   LIN {X -3.366, Y 22.640, Z 44.200}
   LaserEnd_Ext()
   LIN {X 4.267, Y 22.640, Z 44.200}
   LaserStart_Ext()
   LIN {X 6.316, Y 22.640, Z 44.200}
   LaserEnd_Ext()
   LIN {X 6.105, Y 23.640, Z 44.200}
   LaserStart_Ext()
   LIN {X 4.185, Y 23.640, Z 44.200}
   LaserEnd_Ext()
   LIN {X -3.448, Y 23.640, Z 44.200}
   LaserStart_Ext()
   LIN {X -5.428, Y 23.640, Z 44.200}
   LaserEnd_Ext()
   LIN {X -5.387, Y 24.640, Z 44.200}
   LaserStart_Ext()
   LIN {X -3.576, Y 24.640, Z 44.200}
   LaserEnd_Ext()
   LIN {X 4.102, Y 24.640, Z 44.200}
   LaserStart_Ext()
   LIN {X 5.868, Y 24.640, Z 44.200}
   LaserEnd_Ext()
   LIN {X 5.630, Y 25.640, Z 44.200}
   LaserStart_Ext()
   LIN {X 4.020, Y 25.640, Z 44.200}
   LaserEnd_Ext()
   LIN {X -3.712, Y 25.640, Z 44.200}
   LaserStart_Ext()
   LIN {X -5.345, Y 25.640, Z 44.200}
   LaserEnd_Ext()
   LIN {X -5.304, Y 26.640, Z 44.200}
   LaserStart_Ext()
   LIN {X -3.861, Y 26.640, Z 44.200}
   LaserEnd_Ext()
   LIN {X 3.938, Y 26.640, Z 44.200}
   LaserStart_Ext()
   LIN {X 5.393, Y 26.640, Z 44.200}
   LaserEnd_Ext()
   LIN {X 5.155, Y 27.640, Z 44.200}
   LaserStart_Ext()
   LIN {X 3.855, Y 27.640, Z 44.200}
   LaserEnd_Ext()
   LIN {X -4.010, Y 27.640, Z 44.200}
   LaserStart_Ext()
   LIN {X -5.263, Y 27.640, Z 44.200}
   LaserEnd_Ext()
   LIN {X -5.222, Y 28.640, Z 44.200}
   LaserStart_Ext()
   LIN {X -4.204, Y 28.640, Z 44.200}
   LaserEnd_Ext()
   LIN {X 3.773, Y 28.640, Z 44.200}
   LaserStart_Ext()
   LIN {X 4.911, Y 28.640, Z 44.200}
   LaserEnd_Ext()
   LIN {X 4.626, Y 29.640, Z 44.200}
   LaserStart_Ext()
   LIN {X 3.690, Y 29.640, Z 44.200}
   LaserEnd_Ext()
   LIN {X -4.407, Y 29.640, Z 44.200}
   LaserStart_Ext()
   LIN {X -5.180, Y 29.640, Z 44.200}
   LaserEnd_Ext()
   LIN {X -5.139, Y 30.640, Z 44.200}
   LaserStart_Ext()
   LIN {X -4.596, Y 30.640, Z 44.200}
   LaserEnd_Ext()
   LIN {X 3.608, Y 30.640, Z 44.200}
   LaserStart_Ext()
   LIN {X 4.336, Y 30.640, Z 44.200}
   LaserEnd_Ext()
   LIN {X 4.045, Y 31.640, Z 44.200}
   LaserStart_Ext()
   LIN {X 3.526, Y 31.640, Z 44.200}
   LaserEnd_Ext()
   LIN {X -4.818, Y 31.640, Z 44.200}
   LaserStart_Ext()
   LIN {X -5.098, Y 31.640, Z 44.200}
   LaserEnd_Ext()
   LIN {X 3.443, Y 32.640, Z 44.200}
   LaserStart_Ext()
   LIN {X 3.755, Y 32.640, Z 44.200}
   LaserEnd_Ext()
   LIN {X 3.446, Y 33.640, Z 44.200}
   LaserStart_Ext()
   LIN {X 3.361, Y 33.640, Z 44.200}
   LaserEnd_Ext()
   LIN {X -4.883, Y 40.640, Z 44.200}
   LaserStart_Ext()
   LIN {X -4.510, Y 40.640, Z 44.200}
   LaserEnd_Ext()
   LIN {X -1.332, Y 41.640, Z 44.200}
   LaserStart_Ext()
   LIN {X -4.514, Y 41.640, Z 44.200}
   LaserEnd_Ext()
   LIN {X -3.132, Y 42.640, Z 44.200}
   LaserStart_Ext()
   LIN {X -0.665, Y 42.640, Z 44.200}
   LaserEnd_Ext()
   LIN {X -6.671, Y -21.178, Z 45.050}
   LaserStart_Ext()
   LIN {X -6.610, Y -21.017, Z 45.050} C_DIS
   LIN {X -5.679, Y -18.475, Z 45.050} C_DIS
   LIN {X -4.713, Y -17.579, Z 45.050} C_DIS
   LIN {X -4.214, Y -17.153, Z 45.050} C_DIS
   LIN {X -3.553, Y -16.965, Z 45.050} C_DIS
   LIN {X -1.903, Y -16.452, Z 45.050} C_DIS
   LIN {X 0.145, Y -16.770, Z 45.050} C_DIS
   LIN {X 0.270, Y -16.853, Z 45.050} C_DIS
   LIN {X 1.918, Y -17.941, Z 45.050} C_DIS
   LIN {X 3.157, Y -20.130, Z 45.050} C_DIS
   LIN {X 3.247, Y -22.329, Z 45.050} C_DIS
   LIN {X 2.840, Y -23.310, Z 45.050} C_DIS
   LIN {X 2.329, Y -24.417, Z 45.050} C_DIS
   LIN {X 1.031, Y -25.558, Z 45.050} C_DIS
   LIN {X 0.668, Y -25.856, Z 45.050} C_DIS
   LIN {X -0.475, Y -26.166, Z 45.050} C_DIS
   LIN {X -1.451, Y -26.443, Z 45.050} C_DIS
   LIN {X -1.877, Y -26.384, Z 45.050} C_DIS
   LIN {X -3.505, Y -26.122, Z 45.050} C_DIS
   LIN {X -5.111, Y -25.071, Z 45.050} C_DIS
   LIN {X -5.233, Y -24.991, Z 45.050} C_DIS
   LIN {X -5.333, Y -24.835, Z 45.050} C_DIS
   LIN {X -6.364, Y -23.242, Z 45.050} C_DIS
   LIN {X -6.654, Y -21.290, Z 45.050} C_DIS
   LIN {X -6.671, Y -21.178, Z 45.050}
   LaserEnd_Ext()
   LIN {X 2.040, Y 40.494, Z 45.050}
   LaserStart_Ext()
   LIN {X 1.604, Y 41.595, Z 45.050} C_DIS
   LIN {X 0.827, Y 42.817, Z 45.050} C_DIS
   LIN {X -0.621, Y 43.824, Z 45.050} C_DIS
   LIN {X -1.693, Y 44.003, Z 45.050} C_DIS
   LIN {X -2.344, Y 44.109, Z 45.050} C_DIS
   LIN {X -4.381, Y 43.298, Z 45.050} C_DIS
   LIN {X -4.665, Y 43.190, Z 45.050} C_DIS
   LIN {X -5.200, Y 42.535, Z 45.050} C_DIS
   LIN {X -5.616, Y 42.020, Z 45.050} C_DIS
   LIN {X -5.782, Y 41.406, Z 45.050} C_DIS
   LIN {X -6.083, Y 40.281, Z 45.050} C_DIS
   LIN {X -6.024, Y 39.918, Z 45.050} C_DIS
   LIN {X -5.867, Y 38.846, Z 45.050} C_DIS
   LIN {X -5.515, Y 37.770, Z 45.050} C_DIS
   LIN {X -5.478, Y 37.657, Z 45.050} C_DIS
   LIN {X -5.400, Y 37.403, Z 45.050} C_DIS
   LIN {X -5.004, Y 36.129, Z 45.050} C_DIS
   LIN {X -4.447, Y 34.142, Z 45.050} C_DIS
   LIN {X -4.364, Y 33.846, Z 45.050} C_DIS
   LIN {X -4.275, Y 33.476, Z 45.050} C_DIS
   LIN {X -3.760, Y 31.370, Z 45.050} C_DIS
   LIN {X -3.599, Y 30.520, Z 45.050} C_DIS
   LIN {X -3.113, Y 28.175, Z 45.050} C_DIS
   LIN {X -2.524, Y 24.212, Z 45.050} C_DIS
   LIN {X -2.413, Y 23.341, Z 45.050} C_DIS
   LIN {X -2.410, Y 22.832, Z 45.050} C_DIS
   LIN {X -1.992, Y 12.633, Z 45.050} C_DIS
   LIN {X -2.507, Y 7.770, Z 45.050} C_DIS
   LIN {X -2.774, Y 4.413, Z 45.050} C_DIS
   LIN {X -2.802, Y 4.238, Z 45.050} C_DIS
   LIN {X -3.922, Y -1.528, Z 45.050} C_DIS
   LIN {X -4.521, Y -3.749, Z 45.050} C_DIS
   LIN {X -5.169, Y -6.114, Z 45.050} C_DIS
   LIN {X -5.915, Y -8.275, Z 45.050} C_DIS
   LIN {X -6.675, Y -10.509, Z 45.050} C_DIS
   LIN {X -7.437, Y -12.386, Z 45.050} C_DIS
   LIN {X -8.086, Y -13.961, Z 45.050} C_DIS
   LIN {X -9.001, Y -15.896, Z 45.050} C_DIS
   LIN {X -9.722, Y -17.441, Z 45.050} C_DIS
   LIN {X -10.005, Y -18.403, Z 45.050} C_DIS
   LIN {X -10.631, Y -20.479, Z 45.050} C_DIS
   LIN {X -10.320, Y -23.787, Z 45.050} C_DIS
   LIN {X -10.287, Y -24.174, Z 45.050} C_DIS
   LIN {X -10.044, Y -24.611, Z 45.050} C_DIS
   LIN {X -8.449, Y -27.442, Z 45.050} C_DIS
   LIN {X -7.017, Y -28.613, Z 45.050} C_DIS
   LIN {X -6.195, Y -29.276, Z 45.050} C_DIS
   LIN {X -5.563, Y -29.496, Z 45.050} C_DIS
   LIN {X -2.915, Y -30.379, Z 45.050} C_DIS
   LIN {X -0.191, Y -30.129, Z 45.050} C_DIS
   LIN {X 1.018, Y -30.030, Z 45.050} C_DIS
   LIN {X 3.540, Y -28.664, Z 45.050} C_DIS
   LIN {X 3.985, Y -28.426, Z 45.050} C_DIS
   LIN {X 4.171, Y -28.214, Z 45.050} C_DIS
   LIN {X 5.934, Y -26.228, Z 45.050} C_DIS
   LIN {X 6.828, Y -24.050, Z 45.050} C_DIS
   LIN {X 7.136, Y -23.314, Z 45.050} C_DIS
   LIN {X 7.378, Y -22.094, Z 45.050} C_DIS
   LIN {X 7.781, Y -20.115, Z 45.050} C_DIS
   LIN {X 8.099, Y -18.306, Z 45.050} C_DIS
   LIN {X 8.287, Y -17.198, Z 45.050} C_DIS
   LIN {X 8.496, Y -15.692, Z 45.050} C_DIS
   LIN {X 8.821, Y -13.430, Z 45.050} C_DIS
   LIN {X 9.039, Y -11.387, Z 45.050} C_DIS
   LIN {X 9.307, Y -8.680, Z 45.050} C_DIS
   LIN {X 9.533, Y -4.472, Z 45.050} C_DIS
   LIN {X 9.615, Y -3.097, Z 45.050} C_DIS
   LIN {X 9.614, Y -1.693, Z 45.050} C_DIS
   LIN {X 9.577, Y 4.772, Z 45.050} C_DIS
   LIN {X 9.079, Y 9.376, Z 45.050} C_DIS
   LIN {X 8.618, Y 14.785, Z 45.050} C_DIS
   LIN {X 7.738, Y 20.619, Z 45.050} C_DIS
   LIN {X 6.990, Y 24.194, Z 45.050} C_DIS
   LIN {X 6.003, Y 28.349, Z 45.050} C_DIS
   LIN {X 5.310, Y 30.781, Z 45.050} C_DIS
   LIN {X 4.593, Y 33.246, Z 45.050} C_DIS
   LIN {X 4.021, Y 34.987, Z 45.050} C_DIS
   LIN {X 3.789, Y 35.696, Z 45.050} C_DIS
   LIN {X 3.724, Y 35.896, Z 45.050} C_DIS
   LIN {X 3.403, Y 36.808, Z 45.050} C_DIS
   LIN {X 2.943, Y 38.106, Z 45.050} C_DIS
   LIN {X 2.431, Y 39.464, Z 45.050} C_DIS
   LIN {X 2.153, Y 40.206, Z 45.050} C_DIS
   LIN {X 2.040, Y 40.494, Z 45.050}
   LaserEnd_Ext()
   LIN {X 8.602, Y 0.379, Z 45.050}
   LaserStart_Ext()
   LIN {X 8.602, Y -3.288, Z 45.050}
   LaserEnd_Ext()
   LIN {X 7.602, Y -14.881, Z 45.050}
   LaserStart_Ext()
   LIN {X 7.602, Y 14.818, Z 45.050}
   LaserEnd_Ext()
   LIN {X 6.602, Y 21.165, Z 45.050}
   LaserStart_Ext()
   LIN {X 6.602, Y -20.894, Z 45.050}
   LaserEnd_Ext()
   LIN {X 5.602, Y -24.403, Z 45.050}
   LaserStart_Ext()
   LIN {X 5.602, Y 25.712, Z 45.050}
   LaserEnd_Ext()
   LIN {X 4.602, Y 29.617, Z 45.050}
   LaserStart_Ext()
   LIN {X 4.602, Y -26.222, Z 45.050}
   LaserEnd_Ext()
   LIN {X 3.602, Y -27.349, Z 45.050}
   LaserStart_Ext()
   LIN {X 3.602, Y -24.045, Z 45.050}
   LaserEnd_Ext()
   LIN {X 3.602, Y -18.886, Z 45.050}
   LaserStart_Ext()
   LIN {X 3.602, Y 33.060, Z 45.050}
   LaserEnd_Ext()
   LIN {X 2.602, Y 36.071, Z 45.050}
   LaserStart_Ext()
   LIN {X 2.602, Y -17.212, Z 45.050}
   LaserEnd_Ext()
   LIN {X 2.602, Y -25.509, Z 45.050}
   LaserStart_Ext()
   LIN {X 2.602, Y -28.034, Z 45.050}
   LaserEnd_Ext()
   LIN {X 1.602, Y -28.576, Z 45.050}
   LaserStart_Ext()
   LIN {X 1.602, Y -26.383, Z 45.050}
   LaserEnd_Ext()
   LIN {X 1.602, Y -16.534, Z 45.050}
   LaserStart_Ext()
   LIN {X 1.602, Y 38.829, Z 45.050}
   LaserEnd_Ext()
   LIN {X 0.602, Y 41.307, Z 45.050}
   LaserStart_Ext()
   LIN {X 0.602, Y -15.881, Z 45.050}
   LaserEnd_Ext()
   LIN {X 0.602, Y -26.910, Z 45.050}
   LaserStart_Ext()
   LIN {X 0.602, Y -29.061, Z 45.050}
   LaserEnd_Ext()
   LIN {X -0.398, Y -29.144, Z 45.050}
   LaserStart_Ext()
   LIN {X -0.398, Y -27.184, Z 45.050}
   LaserEnd_Ext()
   LIN {X -0.398, Y -15.673, Z 45.050}
   LaserStart_Ext()
   LIN {X -0.398, Y 42.457, Z 45.050}
   LaserEnd_Ext()
   LIN {X -1.398, Y 42.940, Z 45.050}
   LaserStart_Ext()
   LIN {X -1.398, Y 22.553, Z 45.050}
   LaserEnd_Ext()
   LIN {X -1.398, Y 8.750, Z 45.050}
   LaserStart_Ext()
   LIN {X -1.398, Y -15.518, Z 45.050}
   LaserEnd_Ext()
   LIN {X -1.398, Y -27.441, Z 45.050}
   LaserStart_Ext()
   LIN {X -1.398, Y -29.235, Z 45.050}
   LaserEnd_Ext()
   LIN {X -2.398, Y -29.327, Z 45.050}
   LaserStart_Ext()
   LIN {X -2.398, Y -27.313, Z 45.050}
   LaserEnd_Ext()
   LIN {X -2.398, Y -15.558, Z 45.050}
   LaserStart_Ext()
   LIN {X -2.398, Y 1.074, Z 45.050}
   LaserEnd_Ext()
   LIN {X -2.398, Y 29.651, Z 45.050}
   LaserStart_Ext()
   LIN {X -2.398, Y 43.011, Z 45.050}
   LaserEnd_Ext()
   LIN {X -3.398, Y 42.613, Z 45.050}
   LaserStart_Ext()
   LIN {X -3.398, Y 34.104, Z 45.050}
   LaserEnd_Ext()
   LIN {X -3.398, Y -3.425, Z 45.050}
   LaserStart_Ext()
   LIN {X -3.398, Y -15.869, Z 45.050}
   LaserEnd_Ext()
   LIN {X -3.398, Y -27.152, Z 45.050}
   LaserStart_Ext()
   LIN {X -3.398, Y -29.164, Z 45.050}
   LaserEnd_Ext()
   LIN {X -4.398, Y -28.831, Z 45.050}
   LaserStart_Ext()
   LIN {X -4.398, Y -26.732, Z 45.050}
   LaserEnd_Ext()
   LIN {X -4.398, Y -16.166, Z 45.050}
   LaserStart_Ext()
   LIN {X -4.398, Y -6.945, Z 45.050}
   LaserEnd_Ext()
   LIN {X -4.398, Y 37.549, Z 45.050}
   LaserStart_Ext()
   LIN {X -4.398, Y 41.937, Z 45.050}
   LaserEnd_Ext()
   LIN {X -5.398, Y -9.861, Z 45.050}
   LaserStart_Ext()
   LIN {X -5.398, Y -16.851, Z 45.050}
   LaserEnd_Ext()
   LIN {X -5.398, Y -26.078, Z 45.050}
   LaserStart_Ext()
   LIN {X -5.398, Y -28.495, Z 45.050}
   LaserEnd_Ext()
   LIN {X -6.398, Y -27.827, Z 45.050}
   LaserStart_Ext()
   LIN {X -6.398, Y -25.029, Z 45.050}
   LaserEnd_Ext()
   LIN {X -6.398, Y -17.782, Z 45.050}
   LaserStart_Ext()
   LIN {X -6.398, Y -12.485, Z 45.050}
   LaserEnd_Ext()
   LIN {X -7.398, Y -14.846, Z 45.050}
   LaserStart_Ext()
   LIN {X -7.398, Y -20.261, Z 45.050}
   LaserEnd_Ext()
   LIN {X -7.398, Y -23.085, Z 45.050}
   LaserStart_Ext()
   LIN {X -7.398, Y -27.010, Z 45.050}
   LaserEnd_Ext()
   LIN {X -8.398, Y -25.496, Z 45.050}
   LaserStart_Ext()
   LIN {X -8.398, Y -16.969, Z 45.050}
   LaserEnd_Ext()
   LIN {X -9.398, Y -19.854, Z 45.050}
   LaserStart_Ext()
   LIN {X -9.398, Y -22.913, Z 45.050}
   LaserEnd_Ext()
   LIN {X 1.960, Y -24.722, Z 45.900}
   LaserStart_Ext()
   LIN {X 0.859, Y -25.740, Z 45.900} C_DIS
   LIN {X 0.131, Y -25.992, Z 45.900} C_DIS
   LIN {X -1.257, Y -26.384, Z 45.900} C_DIS
   LIN {X -3.022, Y -26.140, Z 45.900} C_DIS
   LIN {X -3.417, Y -26.076, Z 45.900} C_DIS
   LIN {X -3.876, Y -25.776, Z 45.900} C_DIS
   LIN {X -5.147, Y -24.949, Z 45.900} C_DIS
   LIN {X -5.859, Y -23.858, Z 45.900} C_DIS
   LIN {X -6.283, Y -23.203, Z 45.900} C_DIS
   LIN {X -6.394, Y -22.456, Z 45.900} C_DIS
   LIN {X -6.594, Y -21.140, Z 45.900} C_DIS
   LIN {X -6.212, Y -20.025, Z 45.900} C_DIS
   LIN {X -5.649, Y -18.489, Z 45.900} C_DIS
   LIN {X -4.633, Y -17.547, Z 45.900} C_DIS
   LIN {X -4.206, Y -17.142, Z 45.900} C_DIS
   LIN {X -3.214, Y -16.835, Z 45.900} C_DIS
   LIN {X -1.819, Y -16.402, Z 45.900} C_DIS
   LIN {X 0.211, Y -16.716, Z 45.900} C_DIS
   LIN {X 1.455, Y -17.532, Z 45.900} C_DIS
   LIN {X 1.986, Y -17.883, Z 45.900} C_DIS
   LIN {X 2.328, Y -18.486, Z 45.900} C_DIS
   LIN {X 3.245, Y -20.093, Z 45.900} C_DIS
   LIN {X 3.304, Y -21.640, Z 45.900} C_DIS
   LIN {X 3.326, Y -22.267, Z 45.900} C_DIS
   LIN {X 2.604, Y -24.007, Z 45.900} C_DIS
   LIN {X 2.488, Y -24.258, Z 45.900} C_DIS
   LIN {X 1.960, Y -24.722, Z 45.900}
   LaserEnd_Ext()
   LIN {X 8.795, Y -13.943, Z 45.900}
   LaserStart_Ext()
   LIN {X 8.879, Y -13.355, Z 45.900} C_DIS
   LIN {X 8.936, Y -12.824, Z 45.900} C_DIS
   LIN {X 9.355, Y -8.600, Z 45.900} C_DIS
   LIN {X 9.607, Y -3.903, Z 45.900} C_DIS
   LIN {X 9.650, Y -2.973, Z 45.900} C_DIS
   LIN {X 9.643, Y -2.795, Z 45.900} C_DIS
   LIN {X 9.599, Y 4.726, Z 45.900} C_DIS
   LIN {X 8.926, Y 10.955, Z 45.900} C_DIS
   LIN {X 8.556, Y 15.295, Z 45.900} C_DIS
   LIN {X 7.850, Y 19.975, Z 45.900} C_DIS
   LIN {X 6.884, Y 24.593, Z 45.900} C_DIS
   LIN {X 6.088, Y 27.947, Z 45.900} C_DIS
   LIN {X 5.080, Y 31.481, Z 45.900} C_DIS
   LIN {X 4.626, Y 33.041, Z 45.900} C_DIS
   LIN {X 3.895, Y 35.264, Z 45.900} C_DIS
   LIN {X 3.703, Y 35.850, Z 45.900} C_DIS
   LIN {X 3.148, Y 37.401, Z 45.900} C_DIS
   LIN {X 2.802, Y 38.378, Z 45.900} C_DIS
   LIN {X 2.517, Y 39.135, Z 45.900} C_DIS
   LIN {X 2.087, Y 40.261, Z 45.900} C_DIS
   LIN {X 1.596, Y 41.494, Z 45.900} C_DIS
   LIN {X 1.533, Y 41.653, Z 45.900} C_DIS
   LIN {X 1.462, Y 41.765, Z 45.900} C_DIS
   LIN {X 0.740, Y 42.893, Z 45.900} C_DIS
   LIN {X -0.457, Y 43.713, Z 45.900} C_DIS
   LIN {X -0.697, Y 43.876, Z 45.900} C_DIS
   LIN {X -1.138, Y 43.947, Z 45.900} C_DIS
   LIN {X -2.420, Y 44.157, Z 45.900} C_DIS
   LIN {X -3.172, Y 43.857, Z 45.900} C_DIS
   LIN {X -4.678, Y 43.283, Z 45.900} C_DIS
   LIN {X -4.976, Y 42.919, Z 45.900} C_DIS
   LIN {X -5.718, Y 41.999, Z 45.900} C_DIS
   LIN {X -5.957, Y 40.949, Z 45.900} C_DIS
   LIN {X -6.153, Y 40.219, Z 45.900} C_DIS
   LIN {X -5.975, Y 39.137, Z 45.900} C_DIS
   LIN {X -5.931, Y 38.886, Z 45.900} C_DIS
   LIN {X -5.871, Y 38.707, Z 45.900} C_DIS
   LIN {X -5.539, Y 37.698, Z 45.900} C_DIS
   LIN {X -5.073, Y 36.204, Z 45.900} C_DIS
   LIN {X -4.417, Y 33.889, Z 45.900} C_DIS
   LIN {X -3.939, Y 31.967, Z 45.900} C_DIS
   LIN {X -3.840, Y 31.561, Z 45.900} C_DIS
   LIN {X -3.815, Y 31.432, Z 45.900} C_DIS
   LIN {X -3.170, Y 28.317, Z 45.900} C_DIS
   LIN {X -2.623, Y 24.638, Z 45.900} C_DIS
   LIN {X -2.489, Y 23.772, Z 45.900} C_DIS
   LIN {X -2.452, Y 23.526, Z 45.900} C_DIS
   LIN {X -2.422, Y 22.999, Z 45.900} C_DIS
   LIN {X -1.997, Y 12.636, Z 45.900} C_DIS
   LIN {X -2.455, Y 8.315, Z 45.900} C_DIS
   LIN {X -2.691, Y 5.332, Z 45.900} C_DIS
   LIN {X -2.765, Y 4.383, Z 45.900} C_DIS
   LIN {X -3.296, Y 1.594, Z 45.900} C_DIS
   LIN {X -3.905, Y -1.539, Z 45.900} C_DIS
   LIN {X -4.915, Y -5.282, Z 45.900} C_DIS
   LIN {X -5.151, Y -6.143, Z 45.900} C_DIS
   LIN {X -5.422, Y -6.931, Z 45.900} C_DIS
   LIN {X -6.655, Y -10.554, Z 45.900} C_DIS
   LIN {X -7.891, Y -13.597, Z 45.900} C_DIS
   LIN {X -8.027, Y -13.927, Z 45.900} C_DIS
   LIN {X -8.218, Y -14.332, Z 45.900} C_DIS
   LIN {X -9.654, Y -17.411, Z 45.900} C_DIS
   LIN {X -10.218, Y -19.327, Z 45.900} C_DIS
   LIN {X -10.557, Y -20.450, Z 45.900} C_DIS
   LIN {X -10.333, Y -22.829, Z 45.900} C_DIS
   LIN {X -10.204, Y -24.144, Z 45.900} C_DIS
   LIN {X -9.343, Y -25.660, Z 45.900} C_DIS
   LIN {X -8.359, Y -27.408, Z 45.900} C_DIS
   LIN {X -7.745, Y -27.910, Z 45.900} C_DIS
   LIN {X -6.100, Y -29.237, Z 45.900} C_DIS
   LIN {X -4.836, Y -29.678, Z 45.900} C_DIS
   LIN {X -2.908, Y -30.320, Z 45.900} C_DIS
   LIN {X -0.925, Y -30.138, Z 45.900} C_DIS
   LIN {X 1.126, Y -29.970, Z 45.900} C_DIS
   LIN {X 3.152, Y -28.872, Z 45.900} C_DIS
   LIN {X 4.010, Y -28.415, Z 45.900} C_DIS
   LIN {X 4.586, Y -27.798, Z 45.900} C_DIS
   LIN {X 5.980, Y -26.227, Z 45.900} C_DIS
   LIN {X 6.568, Y -24.794, Z 45.900} C_DIS
   LIN {X 7.218, Y -23.243, Z 45.900} C_DIS
   LIN {X 7.727, Y -20.674, Z 45.900} C_DIS
   LIN {X 7.855, Y -20.043, Z 45.900} C_DIS
   LIN {X 7.956, Y -19.466, Z 45.900} C_DIS
   LIN {X 8.354, Y -17.124, Z 45.900} C_DIS
   LIN {X 8.795, Y -13.943, Z 45.900}
   LaserEnd_Ext()
   LIN {X -0.488, Y 42.522, Z 45.900}
   LaserStart_Ext()
   LIN {X -3.868, Y 42.522, Z 45.900}
   LaserEnd_Ext()
   LIN {X -4.801, Y 41.522, Z 45.900}
   LaserStart_Ext()
   LIN {X 0.430, Y 41.522, Z 45.900}
   LaserEnd_Ext()
   LIN {X 0.907, Y 40.522, Z 45.900}
   LaserStart_Ext()
   LIN {X -5.036, Y 40.522, Z 45.900}
   LaserEnd_Ext()
   LIN {X -5.025, Y 39.522, Z 45.900}
   LaserStart_Ext()
   LIN {X 1.299, Y 39.522, Z 45.900}
   LaserEnd_Ext()
   LIN {X 1.680, Y 38.522, Z 45.900}
   LaserStart_Ext()
   LIN {X -4.758, Y 38.522, Z 45.900}
   LaserEnd_Ext()
   LIN {X -4.437, Y 37.522, Z 45.900}
   LaserStart_Ext()
   LIN {X 2.045, Y 37.522, Z 45.900}
   LaserEnd_Ext()
   LIN {X 2.401, Y 36.522, Z 45.900}
   LaserStart_Ext()
   LIN {X -4.124, Y 36.522, Z 45.900}
   LaserEnd_Ext()
   LIN {X -3.839, Y 35.522, Z 45.900}
   LaserStart_Ext()
   LIN {X 2.758, Y 35.522, Z 45.900}
   LaserEnd_Ext()
   LIN {X 3.087, Y 34.522, Z 45.900}
   LaserStart_Ext()
   LIN {X -3.556, Y 34.522, Z 45.900}
   LaserEnd_Ext()
   LIN {X -3.295, Y 33.522, Z 45.900}
   LaserStart_Ext()
   LIN {X 3.415, Y 33.522, Z 45.900}
   LaserEnd_Ext()
   LIN {X 3.736, Y 32.522, Z 45.900}
   LaserStart_Ext()
   LIN {X -3.046, Y 32.522, Z 45.900}
   LaserEnd_Ext()
   LIN {X -2.813, Y 31.522, Z 45.900}
   LaserStart_Ext()
   LIN {X 4.026, Y 31.522, Z 45.900}
   LaserEnd_Ext()
   LIN {X 4.313, Y 30.522, Z 45.900}
   LaserStart_Ext()
   LIN {X -2.605, Y 30.522, Z 45.900}
   LaserEnd_Ext()
   LIN {X -2.398, Y 29.522, Z 45.900}
   LaserStart_Ext()
   LIN {X 4.599, Y 29.522, Z 45.900}
   LaserEnd_Ext()
   LIN {X 4.884, Y 28.522, Z 45.900}
   LaserStart_Ext()
   LIN {X -2.191, Y 28.522, Z 45.900}
   LaserEnd_Ext()
   LIN {X -2.041, Y 27.522, Z 45.900}
   LaserStart_Ext()
   LIN {X 5.161, Y 27.522, Z 45.900}
   LaserEnd_Ext()
   LIN {X 5.398, Y 26.522, Z 45.900}
   LaserStart_Ext()
   LIN {X -1.892, Y 26.522, Z 45.900}
   LaserEnd_Ext()
   LIN {X -1.743, Y 25.522, Z 45.900}
   LaserStart_Ext()
   LIN {X 5.636, Y 25.522, Z 45.900}
   LaserEnd_Ext()
   LIN {X 5.873, Y 24.522, Z 45.900}
   LaserStart_Ext()
   LIN {X -1.593, Y 24.522, Z 45.900}
   LaserEnd_Ext()
   LIN {X -1.450, Y 23.522, Z 45.900}
   LaserStart_Ext()
   LIN {X 6.087, Y 23.522, Z 45.900}
   LaserEnd_Ext()
   LIN {X 6.296, Y 22.522, Z 45.900}
   LaserStart_Ext()
   LIN {X -1.401, Y 22.522, Z 45.900}
   LaserEnd_Ext()
   LIN {X -1.360, Y 21.522, Z 45.900}
   LaserStart_Ext()
   LIN {X 6.505, Y 21.522, Z 45.900}
   LaserEnd_Ext()
   LIN {X 6.714, Y 20.522, Z 45.900}
   LaserStart_Ext()
   LIN {X -1.319, Y 20.522, Z 45.900}
   LaserEnd_Ext()
   LIN {X -1.278, Y 19.522, Z 45.900}
   LaserStart_Ext()
   LIN {X 6.907, Y 19.522, Z 45.900}
   LaserEnd_Ext()
   LIN {X 7.058, Y 18.522, Z 45.900}
   LaserStart_Ext()
   LIN {X -1.237, Y 18.522, Z 45.900}
   LaserEnd_Ext()
   LIN {X -1.196, Y 17.522, Z 45.900}
   LaserStart_Ext()
   LIN {X 7.209, Y 17.522, Z 45.900}
   LaserEnd_Ext()
   LIN {X 7.360, Y 16.522, Z 45.900}
   LaserStart_Ext()
   LIN {X -1.155, Y 16.522, Z 45.900}
   LaserEnd_Ext()
   LIN {X -1.114, Y 15.522, Z 45.900}
   LaserStart_Ext()
   LIN {X 7.511, Y 15.522, Z 45.900}
   LaserEnd_Ext()
   LIN {X 7.619, Y 14.522, Z 45.900}
   LaserStart_Ext()
   LIN {X -1.073, Y 14.522, Z 45.900}
   LaserEnd_Ext()
   LIN {X -1.033, Y 13.522, Z 45.900}
   LaserStart_Ext()
   LIN {X 7.704, Y 13.522, Z 45.900}
   LaserEnd_Ext()
   LIN {X 7.789, Y 12.522, Z 45.900}
   LaserStart_Ext()
   LIN {X -1.004, Y 12.522, Z 45.900}
   LaserEnd_Ext()
   LIN {X -1.110, Y 11.522, Z 45.900}
   LaserStart_Ext()
   LIN {X 7.874, Y 11.522, Z 45.900}
   LaserEnd_Ext()
   LIN {X 7.967, Y 10.522, Z 45.900}
   LaserStart_Ext()
   LIN {X -1.215, Y 10.522, Z 45.900}
   LaserEnd_Ext()
   LIN {X -1.321, Y 9.522, Z 45.900}
   LaserStart_Ext()
   LIN {X 8.075, Y 9.522, Z 45.900}
   LaserEnd_Ext()
   LIN {X 8.183, Y 8.522, Z 45.900}
   LaserStart_Ext()
   LIN {X -1.427, Y 8.522, Z 45.900}
   LaserEnd_Ext()
   LIN {X -1.515, Y 7.522, Z 45.900}
   LaserStart_Ext()
   LIN {X 8.291, Y 7.522, Z 45.900}
   LaserEnd_Ext()
   LIN {X 8.399, Y 6.522, Z 45.900}
   LaserStart_Ext()
   LIN {X -1.594, Y 6.522, Z 45.900}
   LaserEnd_Ext()
   LIN {X -1.673, Y 5.522, Z 45.900}
   LaserStart_Ext()
   LIN {X 8.507, Y 5.522, Z 45.900}
   LaserEnd_Ext()
   LIN {X 8.600, Y 4.522, Z 45.900}
   LaserStart_Ext()
   LIN {X -1.751, Y 4.522, Z 45.900}
   LaserEnd_Ext()
   LIN {X -1.911, Y 3.522, Z 45.900}
   LaserStart_Ext()
   LIN {X 8.606, Y 3.522, Z 45.900}
   LaserEnd_Ext()
   LIN {X 8.612, Y 2.522, Z 45.900}
   LaserStart_Ext()
   LIN {X -2.102, Y 2.522, Z 45.900}
   LaserEnd_Ext()
   LIN {X -2.292, Y 1.522, Z 45.900}
   LaserStart_Ext()
   LIN {X 8.618, Y 1.522, Z 45.900}
   LaserEnd_Ext()
   LIN {X 8.624, Y 0.522, Z 45.900}
   LaserStart_Ext()
   LIN {X -2.486, Y 0.522, Z 45.900}
   LaserEnd_Ext()
   LIN {X -2.680, Y -0.478, Z 45.900}
   LaserStart_Ext()
   LIN {X 8.629, Y -0.478, Z 45.900}
   LaserEnd_Ext()
   LIN {X 8.635, Y -1.478, Z 45.900}
   LaserStart_Ext()
   LIN {X -2.875, Y -1.478, Z 45.900}
   LaserEnd_Ext()
   LIN {X -3.123, Y -2.478, Z 45.900}
   LaserStart_Ext()
   LIN {X 8.641, Y -2.478, Z 45.900}
   LaserEnd_Ext()
   LIN {X 8.625, Y -3.478, Z 45.900}
   LaserStart_Ext()
   LIN {X -3.393, Y -3.478, Z 45.900}
   LaserEnd_Ext()
   LIN {X -3.662, Y -4.478, Z 45.900}
   LaserStart_Ext()
   LIN {X 8.575, Y -4.478, Z 45.900}
   LaserEnd_Ext()
   LIN {X 8.521, Y -5.478, Z 45.900}
   LaserStart_Ext()
   LIN {X -3.932, Y -5.478, Z 45.900}
   LaserEnd_Ext()
   LIN {X -4.208, Y -6.478, Z 45.900}
   LaserStart_Ext()
   LIN {X 8.467, Y -6.478, Z 45.900}
   LaserEnd_Ext()
   LIN {X 8.413, Y -7.478, Z 45.900}
   LaserStart_Ext()
   LIN {X -4.552, Y -7.478, Z 45.900}
   LaserEnd_Ext()
   LIN {X -4.892, Y -8.478, Z 45.900}
   LaserStart_Ext()
   LIN {X 8.360, Y -8.478, Z 45.900}
   LaserEnd_Ext()
   LIN {X 8.263, Y -9.478, Z 45.900}
   LaserStart_Ext()
   LIN {X -5.233, Y -9.478, Z 45.900}
   LaserEnd_Ext()
   LIN {X -5.573, Y -10.478, Z 45.900}
   LaserStart_Ext()
   LIN {X 8.164, Y -10.478, Z 45.900}
   LaserEnd_Ext()
   LIN {X 8.064, Y -11.478, Z 45.900}
   LaserStart_Ext()
   LIN {X -5.951, Y -11.478, Z 45.900}
   LaserEnd_Ext()
   LIN {X -6.357, Y -12.478, Z 45.900}
   LaserStart_Ext()
   LIN {X 7.965, Y -12.478, Z 45.900}
   LaserEnd_Ext()
   LIN {X 7.851, Y -13.478, Z 45.900}
   LaserStart_Ext()
   LIN {X -6.763, Y -13.478, Z 45.900}
   LaserEnd_Ext()
   LIN {X -7.181, Y -14.478, Z 45.900}
   LaserStart_Ext()
   LIN {X 7.711, Y -14.478, Z 45.900}
   LaserEnd_Ext()
   LIN {X 7.572, Y -15.478, Z 45.900}
   LaserStart_Ext()
   LIN {X -1.248, Y -15.478, Z 45.900}
   LaserEnd_Ext()
   LIN {X -2.218, Y -15.478, Z 45.900}
   LaserStart_Ext()
   LIN {X -7.650, Y -15.478, Z 45.900}
   LaserEnd_Ext()
   LIN {X -8.116, Y -16.478, Z 45.900}
   LaserStart_Ext()
   LIN {X -4.959, Y -16.478, Z 45.900}
   LaserEnd_Ext()
   LIN {X 1.672, Y -16.478, Z 45.900}
   LaserStart_Ext()
   LIN {X 7.434, Y -16.478, Z 45.900}
   LaserEnd_Ext()
   LIN {X 7.280, Y -17.478, Z 45.900}
   LaserStart_Ext()
   LIN {X 2.907, Y -17.478, Z 45.900}
   LaserEnd_Ext()
   LIN {X -6.030, Y -17.478, Z 45.900}
   LaserStart_Ext()
   LIN {X -8.583, Y -17.478, Z 45.900}
   LaserEnd_Ext()
   LIN {X -8.926, Y -18.478, Z 45.900}
   LaserStart_Ext()
   LIN {X -6.710, Y -18.478, Z 45.900}
   LaserEnd_Ext()
   LIN {X 3.475, Y -18.478, Z 45.900}
   LaserStart_Ext()
   LIN {X 7.110, Y -18.478, Z 45.900}
   LaserEnd_Ext()
   LIN {X 6.939, Y -19.478, Z 45.900}
   LaserStart_Ext()
   LIN {X 4.045, Y -19.478, Z 45.900}
   LaserEnd_Ext()
   LIN {X -7.076, Y -19.478, Z 45.900}
   LaserStart_Ext()
   LIN {X -9.220, Y -19.478, Z 45.900}
   LaserEnd_Ext()
   LIN {X -9.521, Y -20.478, Z 45.900}
   LaserStart_Ext()
   LIN {X -7.425, Y -20.478, Z 45.900}
   LaserEnd_Ext()
   LIN {X 4.260, Y -20.478, Z 45.900}
   LaserStart_Ext()
   LIN {X 6.746, Y -20.478, Z 45.900}
   LaserEnd_Ext()
   LIN {X 6.548, Y -21.478, Z 45.900}
   LaserStart_Ext()
   LIN {X 4.299, Y -21.478, Z 45.900}
   LaserEnd_Ext()
   LIN {X -7.554, Y -21.478, Z 45.900}
   LaserStart_Ext()
   LIN {X -9.456, Y -21.478, Z 45.900}
   LaserEnd_Ext()
   LIN {X -9.362, Y -22.478, Z 45.900}
   LaserStart_Ext()
   LIN {X -7.402, Y -22.478, Z 45.900}
   LaserEnd_Ext()
   LIN {X 4.302, Y -22.478, Z 45.900}
   LaserStart_Ext()
   LIN {X 6.350, Y -22.478, Z 45.900}
   LaserEnd_Ext()
   LIN {X 6.035, Y -23.478, Z 45.900}
   LaserStart_Ext()
   LIN {X 3.906, Y -23.478, Z 45.900}
   LaserEnd_Ext()
   LIN {X -7.243, Y -23.478, Z 45.900}
   LaserStart_Ext()
   LIN {X -9.265, Y -23.478, Z 45.900}
   LaserEnd_Ext()
   LIN {X -8.864, Y -24.478, Z 45.900}
   LaserStart_Ext()
   LIN {X -6.648, Y -24.478, Z 45.900}
   LaserEnd_Ext()
   LIN {X 3.488, Y -24.478, Z 45.900}
   LaserStart_Ext()
   LIN {X 5.617, Y -24.478, Z 45.900}
   LaserEnd_Ext()
   LIN {X 5.206, Y -25.478, Z 45.900}
   LaserStart_Ext()
   LIN {X 2.615, Y -25.478, Z 45.900}
   LaserEnd_Ext()
   LIN {X -5.996, Y -25.478, Z 45.900}
   LaserStart_Ext()
   LIN {X -8.298, Y -25.478, Z 45.900}
   LaserEnd_Ext()
   LIN {X -7.735, Y -26.478, Z 45.900}
   LaserStart_Ext()
   LIN {X -4.630, Y -26.478, Z 45.900}
   LaserEnd_Ext()
   LIN {X 1.533, Y -26.478, Z 45.900}
   LaserStart_Ext()
   LIN {X 4.420, Y -26.478, Z 45.900}
   LaserEnd_Ext()
   LIN {X 3.517, Y -27.478, Z 45.900}
   LaserStart_Ext()
   LIN {X -6.687, Y -27.478, Z 45.900}
   LaserEnd_Ext()
   LIN {X -5.238, Y -28.478, Z 45.900}
   LaserStart_Ext()
   LIN {X 1.781, Y -28.478, Z 45.900}
   LaserEnd_Ext()
   LIN {X -0.790, Y -26.249, Z 46.750}
   LaserStart_Ext()
   LIN {X -1.064, Y -26.326, Z 46.750} C_DIS
   LIN {X -1.646, Y -26.246, Z 46.750} C_DIS
   LIN {X -3.329, Y -26.031, Z 46.750} C_DIS
   LIN {X -4.112, Y -25.525, Z 46.750} C_DIS
   LIN {X -5.062, Y -24.908, Z 46.750} C_DIS
   LIN {X -5.786, Y -23.797, Z 46.750} C_DIS
   LIN {X -6.201, Y -23.164, Z 46.750} C_DIS
   LIN {X -6.302, Y -22.521, Z 46.750} C_DIS
   LIN {X -6.518, Y -21.102, Z 46.750} C_DIS
   LIN {X -5.725, Y -18.792, Z 46.750} C_DIS
   LIN {X -5.619, Y -18.503, Z 46.750} C_DIS
   LIN {X -5.428, Y -18.326, Z 46.750} C_DIS
   LIN {X -4.122, Y -17.088, Z 46.750} C_DIS
   LIN {X -1.741, Y -16.352, Z 46.750} C_DIS
   LIN {X -1.237, Y -16.428, Z 46.750} C_DIS
   LIN {X 0.277, Y -16.662, Z 46.750} C_DIS
   LIN {X 1.351, Y -17.366, Z 46.750} C_DIS
   LIN {X 2.055, Y -17.824, Z 46.750} C_DIS
   LIN {X 2.655, Y -18.867, Z 46.750} C_DIS
   LIN {X 3.319, Y -20.031, Z 46.750} C_DIS
   LIN {X 3.364, Y -21.206, Z 46.750} C_DIS
   LIN {X 3.253, Y -22.615, Z 46.750} C_DIS
   LIN {X 2.642, Y -24.095, Z 46.750} C_DIS
   LIN {X 1.938, Y -24.811, Z 46.750} C_DIS
   LIN {X 1.084, Y -25.601, Z 46.750} C_DIS
   LIN {X -0.790, Y -26.249, Z 46.750}
   LaserEnd_Ext()
   LIN {X -8.023, Y -14.021, Z 46.750}
   LaserStart_Ext()
   LIN {X -8.376, Y -14.783, Z 46.750} C_DIS
   LIN {X -9.587, Y -17.380, Z 46.750} C_DIS
   LIN {X -10.431, Y -20.250, Z 46.750} C_DIS
   LIN {X -10.482, Y -20.421, Z 46.750} C_DIS
   LIN {X -10.448, Y -20.784, Z 46.750} C_DIS
   LIN {X -10.121, Y -24.114, Z 46.750} C_DIS
   LIN {X -8.447, Y -27.063, Z 46.750} C_DIS
   LIN {X -8.268, Y -27.374, Z 46.750} C_DIS
   LIN {X -7.818, Y -27.735, Z 46.750} C_DIS
   LIN {X -6.005, Y -29.198, Z 46.750} C_DIS
   LIN {X -4.109, Y -29.859, Z 46.750} C_DIS
   LIN {X -2.901, Y -30.261, Z 46.750} C_DIS
   LIN {X -1.659, Y -30.147, Z 46.750} C_DIS
   LIN {X 1.234, Y -29.911, Z 46.750} C_DIS
   LIN {X 2.004, Y -29.493, Z 46.750} C_DIS
   LIN {X 4.010, Y -28.425, Z 46.750} C_DIS
   LIN {X 5.356, Y -26.981, Z 46.750} C_DIS
   LIN {X 6.025, Y -26.226, Z 46.750} C_DIS
   LIN {X 6.308, Y -25.538, Z 46.750} C_DIS
   LIN {X 7.299, Y -23.172, Z 46.750} C_DIS
   LIN {X 7.808, Y -20.603, Z 46.750} C_DIS
   LIN {X 7.929, Y -19.971, Z 46.750} C_DIS
   LIN {X 8.018, Y -19.425, Z 46.750} C_DIS
   LIN {X 8.421, Y -17.051, Z 46.750} C_DIS
   LIN {X 8.829, Y -14.107, Z 46.750} C_DIS
   LIN {X 8.937, Y -13.281, Z 46.750} C_DIS
   LIN {X 9.095, Y -11.618, Z 46.750} C_DIS
   LIN {X 9.402, Y -8.520, Z 46.750} C_DIS
   LIN {X 9.540, Y -5.947, Z 46.750} C_DIS
   LIN {X 9.685, Y -2.789, Z 46.750} C_DIS
   LIN {X 9.662, Y -2.184, Z 46.750} C_DIS
   LIN {X 9.622, Y 4.679, Z 46.750} C_DIS
   LIN {X 8.773, Y 12.535, Z 46.750} C_DIS
   LIN {X 8.495, Y 15.804, Z 46.750} C_DIS
   LIN {X 7.962, Y 19.331, Z 46.750} C_DIS
   LIN {X 6.778, Y 24.991, Z 46.750} C_DIS
   LIN {X 6.172, Y 27.545, Z 46.750} C_DIS
   LIN {X 4.849, Y 32.180, Z 46.750} C_DIS
   LIN {X 4.659, Y 32.836, Z 46.750} C_DIS
   LIN {X 3.769, Y 35.541, Z 46.750} C_DIS
   LIN {X 3.683, Y 35.805, Z 46.750} C_DIS
   LIN {X 3.115, Y 37.392, Z 46.750} C_DIS
   LIN {X 2.706, Y 38.529, Z 46.750} C_DIS
   LIN {X 2.250, Y 39.717, Z 46.750} C_DIS
   LIN {X 2.022, Y 40.315, Z 46.750} C_DIS
   LIN {X 1.890, Y 40.644, Z 46.750} C_DIS
   LIN {X 1.462, Y 41.710, Z 46.750} C_DIS
   LIN {X 0.672, Y 42.939, Z 46.750} C_DIS
   LIN {X -0.773, Y 43.928, Z 46.750} C_DIS
   LIN {X -1.939, Y 44.116, Z 46.750} C_DIS
   LIN {X -2.497, Y 44.204, Z 46.750} C_DIS
   LIN {X -4.064, Y 43.603, Z 46.750} C_DIS
   LIN {X -4.773, Y 43.307, Z 46.750} C_DIS
   LIN {X -5.720, Y 42.092, Z 46.750} C_DIS
   LIN {X -5.835, Y 41.949, Z 46.750} C_DIS
   LIN {X -5.897, Y 41.680, Z 46.750} C_DIS
   LIN {X -6.220, Y 40.247, Z 46.750} C_DIS
   LIN {X -6.119, Y 39.629, Z 46.750} C_DIS
   LIN {X -5.995, Y 38.925, Z 46.750} C_DIS
   LIN {X -5.713, Y 38.073, Z 46.750} C_DIS
   LIN {X -5.601, Y 37.738, Z 46.750} C_DIS
   LIN {X -5.504, Y 37.432, Z 46.750} C_DIS
   LIN {X -5.120, Y 36.212, Z 46.750} C_DIS
   LIN {X -4.541, Y 34.180, Z 46.750} C_DIS
   LIN {X -4.469, Y 33.932, Z 46.750} C_DIS
   LIN {X -4.415, Y 33.717, Z 46.750} C_DIS
   LIN {X -3.893, Y 31.631, Z 46.750} C_DIS
   LIN {X -3.415, Y 29.370, Z 46.750} C_DIS
   LIN {X -3.226, Y 28.460, Z 46.750} C_DIS
   LIN {X -3.094, Y 27.569, Z 46.750} C_DIS
   LIN {X -2.615, Y 24.469, Z 46.750} C_DIS
   LIN {X -2.483, Y 23.590, Z 46.750} C_DIS
   LIN {X -2.373, Y 21.703, Z 46.750} C_DIS
   LIN {X -2.002, Y 12.639, Z 46.750} C_DIS
   LIN {X -2.402, Y 8.860, Z 46.750} C_DIS
   LIN {X -2.609, Y 6.251, Z 46.750} C_DIS
   LIN {X -2.753, Y 4.397, Z 46.750} C_DIS
   LIN {X -3.791, Y -1.050, Z 46.750} C_DIS
   LIN {X -3.888, Y -1.551, Z 46.750} C_DIS
   LIN {X -4.272, Y -2.973, Z 46.750} C_DIS
   LIN {X -5.129, Y -6.166, Z 46.750} C_DIS
   LIN {X -5.366, Y -6.869, Z 46.750} C_DIS
   LIN {X -6.634, Y -10.599, Z 46.750} C_DIS
   LIN {X -7.667, Y -13.141, Z 46.750} C_DIS
   LIN {X -8.023, Y -14.021, Z 46.750}
   LaserEnd_Ext()
   LIN {X -9.280, Y -22.447, Z 46.750}
   LaserStart_Ext()
   LIN {X -9.280, Y -19.881, Z 46.750}
   LaserEnd_Ext()
   LIN {X -8.280, Y -16.943, Z 46.750}
   LaserStart_Ext()
   LIN {X -8.280, Y -25.332, Z 46.750}
   LaserEnd_Ext()
   LIN {X -7.280, Y -26.885, Z 46.750}
   LaserStart_Ext()
   LIN {X -7.280, Y -22.739, Z 46.750}
   LaserEnd_Ext()
   LIN {X -7.280, Y -20.241, Z 46.750}
   LaserStart_Ext()
   LIN {X -7.280, Y -14.796, Z 46.750}
   LaserEnd_Ext()
   LIN {X -6.280, Y -12.383, Z 46.750}
   LaserStart_Ext()
   LIN {X -6.280, Y -17.752, Z 46.750}
   LaserEnd_Ext()
   LIN {X -6.280, Y -24.871, Z 46.750}
   LaserStart_Ext()
   LIN {X -6.280, Y -27.691, Z 46.750}
   LaserEnd_Ext()
   LIN {X -5.280, Y -28.391, Z 46.750}
   LaserStart_Ext()
   LIN {X -5.280, Y -25.959, Z 46.750}
   LaserEnd_Ext()
   LIN {X -5.280, Y -16.807, Z 46.750}
   LaserStart_Ext()
   LIN {X -5.280, Y -9.722, Z 46.750}
   LaserEnd_Ext()
   LIN {X -4.280, Y 42.313, Z 46.750}
   LaserStart_Ext()
   LIN {X -4.280, Y 36.874, Z 46.750}
   LaserEnd_Ext()
   LIN {X -4.280, Y -6.777, Z 46.750}
   LaserStart_Ext()
   LIN {X -4.280, Y -16.090, Z 46.750}
   LaserEnd_Ext()
   LIN {X -4.280, Y -26.607, Z 46.750}
   LaserStart_Ext()
   LIN {X -4.280, Y -28.740, Z 46.750}
   LaserEnd_Ext()
   LIN {X -3.280, Y -29.081, Z 46.750}
   LaserStart_Ext()
   LIN {X -3.280, Y -27.045, Z 46.750}
   LaserEnd_Ext()
   LIN {X -3.280, Y -15.781, Z 46.750}
   LaserStart_Ext()
   LIN {X -3.280, Y -3.135, Z 46.750}
   LaserEnd_Ext()
   LIN {X -3.280, Y 33.301, Z 46.750}
   LaserStart_Ext()
   LIN {X -3.280, Y 42.833, Z 46.750}
   LaserEnd_Ext()
   LIN {X -2.280, Y 43.158, Z 46.750}
   LaserStart_Ext()
   LIN {X -2.280, Y 28.820, Z 46.750}
   LaserEnd_Ext()
   LIN {X -2.280, Y 1.538, Z 46.750}
   LaserStart_Ext()
   LIN {X -2.280, Y -15.472, Z 46.750}
   LaserEnd_Ext()
   LIN {X -2.280, Y -27.173, Z 46.750}
   LaserStart_Ext()
   LIN {X -2.280, Y -29.200, Z 46.750}
   LaserEnd_Ext()
   LIN {X -1.280, Y -29.113, Z 46.750}
   LaserStart_Ext()
   LIN {X -1.280, Y -27.306, Z 46.750}
   LaserEnd_Ext()
   LIN {X -1.280, Y -15.410, Z 46.750}
   LaserStart_Ext()
   LIN {X -1.280, Y 9.962, Z 46.750}
   LaserEnd_Ext()
   LIN {X -1.280, Y 19.444, Z 46.750}
   LaserStart_Ext()
   LIN {X -1.280, Y 42.996, Z 46.750}
   LaserEnd_Ext()
   LIN {X -0.280, Y 42.382, Z 46.750}
   LaserStart_Ext()
   LIN {X -0.280, Y -15.564, Z 46.750}
   LaserEnd_Ext()
   LIN {X -0.280, Y -27.130, Z 46.750}
   LaserStart_Ext()
   LIN {X -0.280, Y -29.031, Z 46.750}
   LaserEnd_Ext()
   LIN {X 0.720, Y -28.949, Z 46.750}
   LaserStart_Ext()
   LIN {X 0.720, Y -26.785, Z 46.750}
   LaserEnd_Ext()
   LIN {X 0.720, Y -15.766, Z 46.750}
   LaserStart_Ext()
   LIN {X 0.720, Y 40.874, Z 46.750}
   LaserEnd_Ext()
   LIN {X 1.720, Y 38.306, Z 46.750}
   LaserStart_Ext()
   LIN {X 1.720, Y -16.412, Z 46.750}
   LaserEnd_Ext()
   LIN {X 1.720, Y -26.371, Z 46.750}
   LaserStart_Ext()
   LIN {X 1.720, Y -28.512, Z 46.750}
   LaserEnd_Ext()
   LIN {X 2.720, Y -27.979, Z 46.750}
   LaserStart_Ext()
   LIN {X 2.720, Y -25.442, Z 46.750}
   LaserEnd_Ext()
   LIN {X 2.720, Y -17.079, Z 46.750}
   LaserStart_Ext()
   LIN {X 2.720, Y 35.528, Z 46.750}
   LaserEnd_Ext()
   LIN {X 3.720, Y 32.483, Z 46.750}
   LaserStart_Ext()
   LIN {X 3.720, Y -18.717, Z 46.750}
   LaserEnd_Ext()
   LIN {X 3.720, Y -24.103, Z 46.750}
   LaserStart_Ext()
   LIN {X 3.720, Y -27.269, Z 46.750}
   LaserEnd_Ext()
   LIN {X 4.720, Y -26.191, Z 46.750}
   LaserStart_Ext()
   LIN {X 4.720, Y 28.989, Z 46.750}
   LaserEnd_Ext()
   LIN {X 5.720, Y 25.119, Z 46.750}
   LaserStart_Ext()
   LIN {X 5.720, Y -24.353, Z 46.750}
   LaserEnd_Ext()
   LIN {X 6.720, Y -20.948, Z 46.750}
   LaserStart_Ext()
   LIN {X 6.720, Y 20.385, Z 46.750}
   LaserEnd_Ext()
   LIN {X 7.720, Y 13.115, Z 46.750}
   LaserStart_Ext()
   LIN {X 7.720, Y -14.822, Z 46.750}
   LaserEnd_Ext()
   LIN {X -6.434, Y -21.115, Z 47.600}
   LaserStart_Ext()
   LIN {X -6.400, Y -20.943, Z 47.600} C_DIS
   LIN {X -5.545, Y -18.457, Z 47.600} C_DIS
   LIN {X -4.509, Y -17.479, Z 47.600} C_DIS
   LIN {X -4.039, Y -17.034, Z 47.600} C_DIS
   LIN {X -1.676, Y -16.302, Z 47.600} C_DIS
   LIN {X 0.274, Y -16.597, Z 47.600} C_DIS
   LIN {X 0.424, Y -16.660, Z 47.600} C_DIS
   LIN {X 2.124, Y -17.766, Z 47.600} C_DIS
   LIN {X 3.111, Y -19.483, Z 47.600} C_DIS
   LIN {X 3.393, Y -19.970, Z 47.600} C_DIS
   LIN {X 3.251, Y -21.001, Z 47.600} C_DIS
   LIN {X 3.074, Y -23.249, Z 47.600} C_DIS
   LIN {X 2.793, Y -23.930, Z 47.600} C_DIS
   LIN {X 1.581, Y -25.165, Z 47.600} C_DIS
   LIN {X 1.304, Y -25.462, Z 47.600} C_DIS
   LIN {X 1.148, Y -25.537, Z 47.600} C_DIS
   LIN {X -0.782, Y -26.244, Z 47.600} C_DIS
   LIN {X -1.919, Y -26.154, Z 47.600} C_DIS
   LIN {X -3.240, Y -25.985, Z 47.600} C_DIS
   LIN {X -4.725, Y -25.027, Z 47.600} C_DIS
   LIN {X -4.976, Y -24.866, Z 47.600} C_DIS
   LIN {X -5.096, Y -24.685, Z 47.600} C_DIS
   LIN {X -6.120, Y -23.125, Z 47.600} C_DIS
   LIN {X -6.434, Y -21.115, Z 47.600}
   LaserEnd_Ext()
   LIN {X -2.513, Y 23.653, Z 47.600}
   LaserStart_Ext()
   LIN {X -2.325, Y 20.407, Z 47.600} C_DIS
   LIN {X -2.007, Y 12.643, Z 47.600} C_DIS
   LIN {X -2.350, Y 9.405, Z 47.600} C_DIS
   LIN {X -2.527, Y 7.170, Z 47.600} C_DIS
   LIN {X -2.741, Y 4.411, Z 47.600} C_DIS
   LIN {X -3.653, Y -0.372, Z 47.600} C_DIS
   LIN {X -3.886, Y -1.633, Z 47.600} C_DIS
   LIN {X -4.196, Y -2.796, Z 47.600} C_DIS
   LIN {X -5.104, Y -6.179, Z 47.600} C_DIS
   LIN {X -5.895, Y -8.530, Z 47.600} C_DIS
   LIN {X -6.614, Y -10.644, Z 47.600} C_DIS
   LIN {X -7.199, Y -12.084, Z 47.600} C_DIS
   LIN {X -8.038, Y -14.161, Z 47.600} C_DIS
   LIN {X -8.871, Y -15.960, Z 47.600} C_DIS
   LIN {X -9.519, Y -17.349, Z 47.600} C_DIS
   LIN {X -10.042, Y -19.125, Z 47.600} C_DIS
   LIN {X -10.408, Y -20.392, Z 47.600} C_DIS
   LIN {X -10.264, Y -21.782, Z 47.600} C_DIS
   LIN {X -10.037, Y -24.084, Z 47.600} C_DIS
   LIN {X -9.073, Y -25.783, Z 47.600} C_DIS
   LIN {X -8.177, Y -27.339, Z 47.600} C_DIS
   LIN {X -5.921, Y -29.149, Z 47.600} C_DIS
   LIN {X -3.382, Y -30.040, Z 47.600} C_DIS
   LIN {X -2.894, Y -30.202, Z 47.600} C_DIS
   LIN {X -2.393, Y -30.156, Z 47.600} C_DIS
   LIN {X -0.223, Y -29.979, Z 47.600} C_DIS
   LIN {X 1.212, Y -29.884, Z 47.600} C_DIS
   LIN {X 1.722, Y -29.653, Z 47.600} C_DIS
   LIN {X 4.009, Y -28.435, Z 47.600} C_DIS
   LIN {X 5.996, Y -26.303, Z 47.600} C_DIS
   LIN {X 6.070, Y -26.227, Z 47.600} C_DIS
   LIN {X 6.153, Y -26.031, Z 47.600} C_DIS
   LIN {X 7.381, Y -23.101, Z 47.600} C_DIS
   LIN {X 7.654, Y -21.719, Z 47.600} C_DIS
   LIN {X 8.003, Y -19.898, Z 47.600} C_DIS
   LIN {X 8.259, Y -18.326, Z 47.600} C_DIS
   LIN {X 8.488, Y -16.977, Z 47.600} C_DIS
   LIN {X 8.720, Y -15.305, Z 47.600} C_DIS
   LIN {X 8.996, Y -13.206, Z 47.600} C_DIS
   LIN {X 9.396, Y -8.982, Z 47.600} C_DIS
   LIN {X 9.449, Y -8.440, Z 47.600} C_DIS
   LIN {X 9.473, Y -7.990, Z 47.600} C_DIS
   LIN {X 9.721, Y -2.604, Z 47.600} C_DIS
   LIN {X 9.680, Y -1.572, Z 47.600} C_DIS
   LIN {X 9.645, Y 4.633, Z 47.600} C_DIS
   LIN {X 8.620, Y 14.114, Z 47.600} C_DIS
   LIN {X 8.433, Y 16.314, Z 47.600} C_DIS
   LIN {X 8.075, Y 18.686, Z 47.600} C_DIS
   LIN {X 6.673, Y 25.389, Z 47.600} C_DIS
   LIN {X 6.256, Y 27.143, Z 47.600} C_DIS
   LIN {X 4.879, Y 31.972, Z 47.600} C_DIS
   LIN {X 4.660, Y 32.735, Z 47.600} C_DIS
   LIN {X 3.733, Y 35.551, Z 47.600} C_DIS
   LIN {X 3.657, Y 35.778, Z 47.600} C_DIS
   LIN {X 3.376, Y 36.552, Z 47.600} C_DIS
   LIN {X 2.644, Y 38.584, Z 47.600} C_DIS
   LIN {X 2.371, Y 39.295, Z 47.600} C_DIS
   LIN {X 1.952, Y 40.378, Z 47.600} C_DIS
   LIN {X 1.466, Y 41.581, Z 47.600} C_DIS
   LIN {X 1.391, Y 41.767, Z 47.600} C_DIS
   LIN {X 1.311, Y 41.891, Z 47.600} C_DIS
   LIN {X 0.593, Y 43.003, Z 47.600} C_DIS
   LIN {X -0.691, Y 43.872, Z 47.600} C_DIS
   LIN {X -0.849, Y 43.979, Z 47.600} C_DIS
   LIN {X -1.222, Y 44.038, Z 47.600} C_DIS
   LIN {X -2.573, Y 44.252, Z 47.600} C_DIS
   LIN {X -3.081, Y 44.057, Z 47.600} C_DIS
   LIN {X -4.917, Y 43.290, Z 47.600} C_DIS
   LIN {X -5.175, Y 42.959, Z 47.600} C_DIS
   LIN {X -5.936, Y 41.925, Z 47.600} C_DIS
   LIN {X -6.195, Y 40.802, Z 47.600} C_DIS
   LIN {X -6.286, Y 40.397, Z 47.600} C_DIS
   LIN {X -6.200, Y 39.873, Z 47.600} C_DIS
   LIN {X -6.059, Y 38.964, Z 47.600} C_DIS
   LIN {X -5.882, Y 38.439, Z 47.600} C_DIS
   LIN {X -5.662, Y 37.778, Z 47.600} C_DIS
   LIN {X -5.289, Y 36.600, Z 47.600} C_DIS
   LIN {X -5.178, Y 36.253, Z 47.600} C_DIS
   LIN {X -5.045, Y 35.795, Z 47.600} C_DIS
   LIN {X -4.521, Y 33.974, Z 47.600} C_DIS
   LIN {X -3.955, Y 31.736, Z 47.600} C_DIS
   LIN {X -3.374, Y 29.038, Z 47.600} C_DIS
   LIN {X -3.210, Y 28.204, Z 47.600} C_DIS
   LIN {X -2.741, Y 25.167, Z 47.600} C_DIS
   LIN {X -2.513, Y 23.653, Z 47.600}
   LaserEnd_Ext()
   LIN {X 2.023, Y -28.360, Z 47.600}
   LaserStart_Ext()
   LIN {X -5.161, Y -28.360, Z 47.600}
   LaserEnd_Ext()
   LIN {X -6.553, Y -27.360, Z 47.600}
   LaserStart_Ext()
   LIN {X 3.644, Y -27.360, Z 47.600}
   LaserEnd_Ext()
   LIN {X 4.576, Y -26.360, Z 47.600}
   LaserStart_Ext()
   LIN {X 1.743, Y -26.360, Z 47.600}
   LaserEnd_Ext()
   LIN {X -4.504, Y -26.360, Z 47.600}
   LaserStart_Ext()
   LIN {X -7.587, Y -26.360, Z 47.600}
   LaserEnd_Ext()
   LIN {X -8.163, Y -25.360, Z 47.600}
   LaserStart_Ext()
   LIN {X -5.849, Y -25.360, Z 47.600}
   LaserEnd_Ext()
   LIN {X 2.791, Y -25.360, Z 47.600}
   LaserStart_Ext()
   LIN {X 5.350, Y -25.360, Z 47.600}
   LaserEnd_Ext()
   LIN {X 5.769, Y -24.360, Z 47.600}
   LaserStart_Ext()
   LIN {X 3.694, Y -24.360, Z 47.600}
   LaserEnd_Ext()
   LIN {X -6.506, Y -24.360, Z 47.600}
   LaserStart_Ext()
   LIN {X -8.731, Y -24.360, Z 47.600}
   LaserEnd_Ext()
   LIN {X -9.104, Y -23.360, Z 47.600}
   LaserStart_Ext()
   LIN {X -7.091, Y -23.360, Z 47.600}
   LaserEnd_Ext()
   LIN {X 4.067, Y -23.360, Z 47.600}
   LaserStart_Ext()
   LIN {X 6.188, Y -23.360, Z 47.600}
   LaserEnd_Ext()
   LIN {X 6.508, Y -22.360, Z 47.600}
   LaserStart_Ext()
   LIN {X 4.147, Y -22.360, Z 47.600}
   LaserEnd_Ext()
   LIN {X -7.252, Y -22.360, Z 47.600}
   LaserStart_Ext()
   LIN {X -9.202, Y -22.360, Z 47.600}
   LaserEnd_Ext()
   LIN {X -9.302, Y -21.360, Z 47.600}
   LaserStart_Ext()
   LIN {X -7.408, Y -21.360, Z 47.600}
   LaserEnd_Ext()
   LIN {X 4.226, Y -21.360, Z 47.600}
   LaserStart_Ext()
   LIN {X 6.705, Y -21.360, Z 47.600}
   LaserEnd_Ext()
   LIN {X 6.896, Y -20.360, Z 47.600}
   LaserStart_Ext()
   LIN {X 4.348, Y -20.360, Z 47.600}
   LaserEnd_Ext()
   LIN {X -7.257, Y -20.360, Z 47.600}
   LaserStart_Ext()
   LIN {X -9.357, Y -20.360, Z 47.600}
   LaserEnd_Ext()
   LIN {X -9.068, Y -19.360, Z 47.600}
   LaserStart_Ext()
   LIN {X -6.913, Y -19.360, Z 47.600}
   LaserEnd_Ext()
   LIN {X 4.195, Y -19.360, Z 47.600}
   LaserStart_Ext()
   LIN {X 7.077, Y -19.360, Z 47.600}
   LaserEnd_Ext()
   LIN {X 7.240, Y -18.360, Z 47.600}
   LaserStart_Ext()
   LIN {X 3.619, Y -18.360, Z 47.600}
   LaserEnd_Ext()
   LIN {X -6.569, Y -18.360, Z 47.600}
   LaserStart_Ext()
   LIN {X -8.774, Y -18.360, Z 47.600}
   LaserEnd_Ext()
   LIN {X -8.421, Y -17.360, Z 47.600}
   LaserStart_Ext()
   LIN {X -5.840, Y -17.360, Z 47.600}
   LaserEnd_Ext()
   LIN {X 3.044, Y -17.360, Z 47.600}
   LaserStart_Ext()
   LIN {X 7.409, Y -17.360, Z 47.600}
   LaserEnd_Ext()
   LIN {X 7.564, Y -16.360, Z 47.600}
   LaserStart_Ext()
   LIN {X 1.797, Y -16.360, Z 47.600}
   LaserEnd_Ext()
   LIN {X -4.782, Y -16.360, Z 47.600}
   LaserStart_Ext()
   LIN {X -7.955, Y -16.360, Z 47.600}
   LaserEnd_Ext()
   LIN {X -7.492, Y -15.360, Z 47.600}
   LaserStart_Ext()
   LIN {X -2.014, Y -15.360, Z 47.600}
   LaserEnd_Ext()
   LIN {X -1.218, Y -15.360, Z 47.600}
   LaserStart_Ext()
   LIN {X 7.702, Y -15.360, Z 47.600}
   LaserEnd_Ext()
   LIN {X 7.835, Y -14.360, Z 47.600}
   LaserStart_Ext()
   LIN {X -7.040, Y -14.360, Z 47.600}
   LaserEnd_Ext()
   LIN {X -6.636, Y -13.360, Z 47.600}
   LaserStart_Ext()
   LIN {X 7.967, Y -13.360, Z 47.600}
   LaserEnd_Ext()
   LIN {X 8.071, Y -12.360, Z 47.600}
   LaserStart_Ext()
   LIN {X -6.232, Y -12.360, Z 47.600}
   LaserEnd_Ext()
   LIN {X -5.826, Y -11.360, Z 47.600}
   LaserStart_Ext()
   LIN {X 8.166, Y -11.360, Z 47.600}
   LaserEnd_Ext()
   LIN {X 8.261, Y -10.360, Z 47.600}
   LaserStart_Ext()
   LIN {X -5.461, Y -10.360, Z 47.600}
   LaserEnd_Ext()
   LIN {X -5.121, Y -9.360, Z 47.600}
   LaserStart_Ext()
   LIN {X 8.355, Y -9.360, Z 47.600}
   LaserEnd_Ext()
   LIN {X 8.452, Y -8.360, Z 47.600}
   LaserStart_Ext()
   LIN {X -4.783, Y -8.360, Z 47.600}
   LaserEnd_Ext()
   LIN {X -4.447, Y -7.360, Z 47.600}
   LaserStart_Ext()
   LIN {X 8.501, Y -7.360, Z 47.600}
   LaserEnd_Ext()
   LIN {X 8.547, Y -6.360, Z 47.600}
   LaserStart_Ext()
   LIN {X -4.117, Y -6.360, Z 47.600}
   LaserEnd_Ext()
   LIN {X -3.849, Y -5.360, Z 47.600}
   LaserStart_Ext()
   LIN {X 8.593, Y -5.360, Z 47.600}
   LaserEnd_Ext()
   LIN {X 8.639, Y -4.360, Z 47.600}
   LaserStart_Ext()
   LIN {X -3.580, Y -4.360, Z 47.600}
   LaserEnd_Ext()
   LIN {X -3.312, Y -3.360, Z 47.600}
   LaserStart_Ext()
   LIN {X 8.685, Y -3.360, Z 47.600}
   LaserEnd_Ext()
   LIN {X 8.711, Y -2.360, Z 47.600}
   LaserStart_Ext()
   LIN {X -3.045, Y -2.360, Z 47.600}
   LaserEnd_Ext()
   LIN {X -2.819, Y -1.360, Z 47.600}
   LaserStart_Ext()
   LIN {X 8.679, Y -1.360, Z 47.600}
   LaserEnd_Ext()
   LIN {X 8.673, Y -0.360, Z 47.600}
   LaserStart_Ext()
   LIN {X -2.632, Y -0.360, Z 47.600}
   LaserEnd_Ext()
   LIN {X -2.442, Y 0.640, Z 47.600}
   LaserStart_Ext()
   LIN {X 8.668, Y 0.640, Z 47.600}
   LaserEnd_Ext()
   LIN {X 8.662, Y 1.640, Z 47.600}
   LaserStart_Ext()
   LIN {X -2.251, Y 1.640, Z 47.600}
   LaserEnd_Ext()
   LIN {X -2.061, Y 2.640, Z 47.600}
   LaserStart_Ext()
   LIN {X 8.656, Y 2.640, Z 47.600}
   LaserEnd_Ext()
   LIN {X 8.650, Y 3.640, Z 47.600}
   LaserStart_Ext()
   LIN {X -1.870, Y 3.640, Z 47.600}
   LaserEnd_Ext()
   LIN {X -1.720, Y 4.640, Z 47.600}
   LaserStart_Ext()
   LIN {X 8.638, Y 4.640, Z 47.600}
   LaserEnd_Ext()
   LIN {X 8.530, Y 5.640, Z 47.600}
   LaserStart_Ext()
   LIN {X -1.643, Y 5.640, Z 47.600}
   LaserEnd_Ext()
   LIN {X -1.565, Y 6.640, Z 47.600}
   LaserStart_Ext()
   LIN {X 8.422, Y 6.640, Z 47.600}
   LaserEnd_Ext()
   LIN {X 8.314, Y 7.640, Z 47.600}
   LaserStart_Ext()
   LIN {X -1.486, Y 7.640, Z 47.600}
   LaserEnd_Ext()
   LIN {X -1.407, Y 8.640, Z 47.600}
   LaserStart_Ext()
   LIN {X 8.206, Y 8.640, Z 47.600}
   LaserEnd_Ext()
   LIN {X 8.098, Y 9.640, Z 47.600}
   LaserStart_Ext()
   LIN {X -1.319, Y 9.640, Z 47.600}
   LaserEnd_Ext()
   LIN {X -1.213, Y 10.640, Z 47.600}
   LaserStart_Ext()
   LIN {X 7.990, Y 10.640, Z 47.600}
   LaserEnd_Ext()
   LIN {X 7.882, Y 11.640, Z 47.600}
   LaserStart_Ext()
   LIN {X -1.107, Y 11.640, Z 47.600}
   LaserEnd_Ext()
   LIN {X -1.009, Y 12.640, Z 47.600}
   LaserStart_Ext()
   LIN {X 7.774, Y 12.640, Z 47.600}
   LaserEnd_Ext()
   LIN {X 7.666, Y 13.640, Z 47.600}
   LaserStart_Ext()
   LIN {X -1.047, Y 13.640, Z 47.600}
   LaserEnd_Ext()
   LIN {X -1.088, Y 14.640, Z 47.600}
   LaserStart_Ext()
   LIN {X 7.572, Y 14.640, Z 47.600}
   LaserEnd_Ext()
   LIN {X 7.487, Y 15.640, Z 47.600}
   LaserStart_Ext()
   LIN {X -1.129, Y 15.640, Z 47.600}
   LaserEnd_Ext()
   LIN {X -1.170, Y 16.640, Z 47.600}
   LaserStart_Ext()
   LIN {X 7.372, Y 16.640, Z 47.600}
   LaserEnd_Ext()
   LIN {X 7.221, Y 17.640, Z 47.600}
   LaserStart_Ext()
   LIN {X -1.211, Y 17.640, Z 47.600}
   LaserEnd_Ext()
   LIN {X -1.252, Y 18.640, Z 47.600}
   LaserStart_Ext()
   LIN {X 7.063, Y 18.640, Z 47.600}
   LaserEnd_Ext()
   LIN {X 6.854, Y 19.640, Z 47.600}
   LaserStart_Ext()
   LIN {X -1.293, Y 19.640, Z 47.600}
   LaserEnd_Ext()
   LIN {X -1.337, Y 20.640, Z 47.600}
   LaserStart_Ext()
   LIN {X 6.644, Y 20.640, Z 47.600}
   LaserEnd_Ext()
   LIN {X 6.435, Y 21.640, Z 47.600}
   LaserStart_Ext()
   LIN {X -1.395, Y 21.640, Z 47.600}
   LaserEnd_Ext()
   LIN {X -1.452, Y 22.640, Z 47.600}
   LaserStart_Ext()
   LIN {X 6.226, Y 22.640, Z 47.600}
   LaserEnd_Ext()
   LIN {X 6.017, Y 23.640, Z 47.600}
   LaserStart_Ext()
   LIN {X -1.510, Y 23.640, Z 47.600}
   LaserEnd_Ext()
   LIN {X -1.650, Y 24.640, Z 47.600}
   LaserStart_Ext()
   LIN {X 5.808, Y 24.640, Z 47.600}
   LaserEnd_Ext()
   LIN {X 5.585, Y 25.640, Z 47.600}
   LaserStart_Ext()
   LIN {X -1.802, Y 25.640, Z 47.600}
   LaserEnd_Ext()
   LIN {X -1.956, Y 26.640, Z 47.600}
   LaserStart_Ext()
   LIN {X 5.348, Y 26.640, Z 47.600}
   LaserEnd_Ext()
   LIN {X 5.075, Y 27.640, Z 47.600}
   LaserStart_Ext()
   LIN {X -2.111, Y 27.640, Z 47.600}
   LaserEnd_Ext()
   LIN {X -2.277, Y 28.640, Z 47.600}
   LaserStart_Ext()
   LIN {X 4.789, Y 28.640, Z 47.600}
   LaserEnd_Ext()
   LIN {X 4.504, Y 29.640, Z 47.600}
   LaserStart_Ext()
   LIN {X -2.481, Y 29.640, Z 47.600}
   LaserEnd_Ext()
   LIN {X -2.695, Y 30.640, Z 47.600}
   LaserStart_Ext()
   LIN {X 4.219, Y 30.640, Z 47.600}
   LaserEnd_Ext()
   LIN {X 3.933, Y 31.640, Z 47.600}
   LaserStart_Ext()
   LIN {X -2.909, Y 31.640, Z 47.600}
   LaserEnd_Ext()
   LIN {X -3.152, Y 32.640, Z 47.600}
   LaserStart_Ext()
   LIN {X 3.638, Y 32.640, Z 47.600}
   LaserEnd_Ext()
   LIN {X 3.309, Y 33.640, Z 47.600}
   LaserStart_Ext()
   LIN {X -3.405, Y 33.640, Z 47.600}
   LaserEnd_Ext()
   LIN {X -3.672, Y 34.640, Z 47.600}
   LaserStart_Ext()
   LIN {X 2.980, Y 34.640, Z 47.600}
   LaserEnd_Ext()
   LIN {X 2.643, Y 35.640, Z 47.600}
   LaserStart_Ext()
   LIN {X -3.960, Y 35.640, Z 47.600}
   LaserEnd_Ext()
   LIN {X -4.251, Y 36.640, Z 47.600}
   LaserStart_Ext()
   LIN {X 2.282, Y 36.640, Z 47.600}
   LaserEnd_Ext()
   LIN {X 1.921, Y 37.640, Z 47.600}
   LaserStart_Ext()
   LIN {X -4.569, Y 37.640, Z 47.600}
   LaserEnd_Ext()
   LIN {X -4.895, Y 38.640, Z 47.600}
   LaserStart_Ext()
   LIN {X 1.552, Y 38.640, Z 47.600}
   LaserEnd_Ext()
   LIN {X 1.165, Y 39.640, Z 47.600}
   LaserStart_Ext()
   LIN {X -5.152, Y 39.640, Z 47.600}
   LaserEnd_Ext()
   LIN {X -5.206, Y 40.640, Z 47.600}
   LaserStart_Ext()
   LIN {X 0.768, Y 40.640, Z 47.600}
   LaserEnd_Ext()
   LIN {X 0.283, Y 41.640, Z 47.600}
   LaserStart_Ext()
   LIN {X -4.904, Y 41.640, Z 47.600}
   LaserEnd_Ext()
   LIN {X -3.879, Y 42.640, Z 47.600}
   LaserStart_Ext()
   LIN {X -0.654, Y 42.640, Z 47.600}
   LaserEnd_Ext()
   LIN {X 2.272, Y -17.845, Z 48.450}
   LaserStart_Ext()
   LIN {X 3.467, Y -19.908, Z 48.450} C_DIS
   LIN {X 2.976, Y -23.464, Z 48.450} C_DIS
   LIN {X 2.955, Y -23.733, Z 48.450} C_DIS
   LIN {X 2.862, Y -23.865, Z 48.450} C_DIS
   LIN {X 1.499, Y -25.326, Z 48.450} C_DIS
   LIN {X 0.569, Y -25.773, Z 48.450} C_DIS
   LIN {X -0.471, Y -26.153, Z 48.450} C_DIS
   LIN {X -3.115, Y -25.944, Z 48.450} C_DIS
   LIN {X -4.891, Y -24.824, Z 48.450} C_DIS
   LIN {X -5.698, Y -23.605, Z 48.450} C_DIS
   LIN {X -6.039, Y -23.086, Z 48.450} C_DIS
   LIN {X -6.148, Y -22.383, Z 48.450} C_DIS
   LIN {X -6.365, Y -21.025, Z 48.450} C_DIS
   LIN {X -5.933, Y -19.774, Z 48.450} C_DIS
   LIN {X -5.458, Y -18.393, Z 48.450} C_DIS
   LIN {X -4.519, Y -17.507, Z 48.450} C_DIS
   LIN {X -3.950, Y -16.977, Z 48.450} C_DIS
   LIN {X -1.610, Y -16.253, Z 48.450} C_DIS
   LIN {X -0.997, Y -16.345, Z 48.450} C_DIS
   LIN {X 0.409, Y -16.553, Z 48.450} C_DIS
   LIN {X 2.057, Y -17.619, Z 48.450} C_DIS
   LIN {X 2.193, Y -17.707, Z 48.450} C_DIS
   LIN {X 2.272, Y -17.845, Z 48.450}
   LaserEnd_Ext()
   LIN {X -9.452, Y -17.318, Z 48.450}
   LaserStart_Ext()
   LIN {X -9.520, Y -17.550, Z 48.450} C_DIS
   LIN {X -10.333, Y -20.363, Z 48.450} C_DIS
   LIN {X -10.014, Y -23.447, Z 48.450} C_DIS
   LIN {X -9.954, Y -24.054, Z 48.450} C_DIS
   LIN {X -9.700, Y -24.503, Z 48.450} C_DIS
   LIN {X -8.086, Y -27.305, Z 48.450} C_DIS
   LIN {X -6.637, Y -28.467, Z 48.450} C_DIS
   LIN {X -5.814, Y -29.118, Z 48.450} C_DIS
   LIN {X -3.145, Y -30.049, Z 48.450} C_DIS
   LIN {X -2.603, Y -30.146, Z 48.450} C_DIS
   LIN {X 0.982, Y -29.908, Z 48.450} C_DIS
   LIN {X 2.813, Y -29.082, Z 48.450} C_DIS
   LIN {X 4.009, Y -28.445, Z 48.450} C_DIS
   LIN {X 5.047, Y -27.330, Z 48.450} C_DIS
   LIN {X 6.105, Y -26.238, Z 48.450} C_DIS
   LIN {X 7.289, Y -23.444, Z 48.450} C_DIS
   LIN {X 7.462, Y -23.031, Z 48.450} C_DIS
   LIN {X 7.501, Y -22.836, Z 48.450} C_DIS
   LIN {X 8.077, Y -19.826, Z 48.450} C_DIS
   LIN {X 8.500, Y -17.227, Z 48.450} C_DIS
   LIN {X 8.555, Y -16.904, Z 48.450} C_DIS
   LIN {X 8.610, Y -16.504, Z 48.450} C_DIS
   LIN {X 9.054, Y -13.131, Z 48.450} C_DIS
   LIN {X 9.383, Y -9.651, Z 48.450} C_DIS
   LIN {X 9.496, Y -8.363, Z 48.450} C_DIS
   LIN {X 9.613, Y -5.551, Z 48.450} C_DIS
   LIN {X 9.757, Y -2.419, Z 48.450} C_DIS
   LIN {X 9.699, Y -0.960, Z 48.450} C_DIS
   LIN {X 9.667, Y 4.586, Z 48.450} C_DIS
   LIN {X 8.467, Y 15.693, Z 48.450} C_DIS
   LIN {X 8.371, Y 16.823, Z 48.450} C_DIS
   LIN {X 8.187, Y 18.042, Z 48.450} C_DIS
   LIN {X 6.567, Y 25.787, Z 48.450} C_DIS
   LIN {X 6.340, Y 26.741, Z 48.450} C_DIS
   LIN {X 5.591, Y 29.368, Z 48.450} C_DIS
   LIN {X 4.576, Y 32.907, Z 48.450} C_DIS
   LIN {X 4.098, Y 34.359, Z 48.450} C_DIS
   LIN {X 3.601, Y 35.836, Z 48.450} C_DIS
   LIN {X 2.972, Y 37.573, Z 48.450} C_DIS
   LIN {X 2.580, Y 38.647, Z 48.450} C_DIS
   LIN {X 2.138, Y 39.781, Z 48.450} C_DIS
   LIN {X 1.881, Y 40.445, Z 48.450} C_DIS
   LIN {X 1.737, Y 40.800, Z 48.450} C_DIS
   LIN {X 1.321, Y 41.823, Z 48.450} C_DIS
   LIN {X 0.581, Y 42.961, Z 48.450} C_DIS
   LIN {X 0.519, Y 43.058, Z 48.450} C_DIS
   LIN {X 0.429, Y 43.118, Z 48.450} C_DIS
   LIN {X -0.925, Y 44.030, Z 48.450} C_DIS
   LIN {X -1.948, Y 44.191, Z 48.450} C_DIS
   LIN {X -2.650, Y 44.299, Z 48.450} C_DIS
   LIN {X -4.285, Y 43.620, Z 48.450} C_DIS
   LIN {X -5.059, Y 43.270, Z 48.450} C_DIS
   LIN {X -6.013, Y 41.932, Z 48.450} C_DIS
   LIN {X -6.353, Y 40.375, Z 48.450} C_DIS
   LIN {X -6.195, Y 39.467, Z 48.450} C_DIS
   LIN {X -6.123, Y 39.003, Z 48.450} C_DIS
   LIN {X -5.944, Y 38.470, Z 48.450} C_DIS
   LIN {X -5.723, Y 37.818, Z 48.450} C_DIS
   LIN {X -5.532, Y 37.222, Z 48.450} C_DIS
   LIN {X -5.235, Y 36.294, Z 48.450} C_DIS
   LIN {X -4.788, Y 34.750, Z 48.450} C_DIS
   LIN {X -4.574, Y 34.017, Z 48.450} C_DIS
   LIN {X -4.387, Y 33.291, Z 48.450} C_DIS
   LIN {X -3.987, Y 31.719, Z 48.450} C_DIS
   LIN {X -3.740, Y 30.635, Z 48.450} C_DIS
   LIN {X -3.565, Y 29.821, Z 48.450} C_DIS
   LIN {X -3.160, Y 27.763, Z 48.450} C_DIS
   LIN {X -2.866, Y 25.864, Z 48.450} C_DIS
   LIN {X -2.543, Y 23.716, Z 48.450} C_DIS
   LIN {X -2.276, Y 19.111, Z 48.450} C_DIS
   LIN {X -2.011, Y 12.646, Z 48.450} C_DIS
   LIN {X -2.297, Y 9.950, Z 48.450} C_DIS
   LIN {X -2.444, Y 8.089, Z 48.450} C_DIS
   LIN {X -2.729, Y 4.425, Z 48.450} C_DIS
   LIN {X -3.366, Y 1.085, Z 48.450} C_DIS
   LIN {X -3.888, Y -1.732, Z 48.450} C_DIS
   LIN {X -4.579, Y -4.332, Z 48.450} C_DIS
   LIN {X -5.079, Y -6.192, Z 48.450} C_DIS
   LIN {X -6.424, Y -10.191, Z 48.450} C_DIS
   LIN {X -6.594, Y -10.688, Z 48.450} C_DIS
   LIN {X -6.731, Y -11.027, Z 48.450} C_DIS
   LIN {X -8.054, Y -14.302, Z 48.450} C_DIS
   LIN {X -9.367, Y -17.137, Z 48.450} C_DIS
   LIN {X -9.452, Y -17.318, Z 48.450}
   LaserEnd_Ext()
   LIN {X 8.602, Y 5.137, Z 48.450}
   LaserStart_Ext()
   LIN {X 8.602, Y -5.790, Z 48.450}
   LaserEnd_Ext()
   LIN {X 7.602, Y -16.496, Z 48.450}
   LaserStart_Ext()
   LIN {X 7.602, Y 14.393, Z 48.450}
   LaserEnd_Ext()
   LIN {X 6.602, Y 20.736, Z 48.450}
   LaserStart_Ext()
   LIN {X 6.602, Y -22.212, Z 48.450}
   LaserEnd_Ext()
   LIN {X 5.602, Y -24.862, Z 48.450}
   LaserStart_Ext()
   LIN {X 5.602, Y 25.517, Z 48.450}
   LaserEnd_Ext()
   LIN {X 4.602, Y 29.189, Z 48.450}
   LaserStart_Ext()
   LIN {X 4.602, Y -26.353, Z 48.450}
   LaserEnd_Ext()
   LIN {X 3.602, Y -27.414, Z 48.450}
   LaserStart_Ext()
   LIN {X 3.602, Y -24.537, Z 48.450}
   LaserEnd_Ext()
   LIN {X 3.602, Y -18.146, Z 48.450}
   LaserStart_Ext()
   LIN {X 3.602, Y 32.666, Z 48.450}
   LaserEnd_Ext()
   LIN {X 2.602, Y 35.659, Z 48.450}
   LaserStart_Ext()
   LIN {X 2.602, Y -16.780, Z 48.450}
   LaserEnd_Ext()
   LIN {X 2.602, Y -25.609, Z 48.450}
   LaserStart_Ext()
   LIN {X 2.602, Y -28.061, Z 48.450}
   LaserEnd_Ext()
   LIN {X 1.602, Y -28.531, Z 48.450}
   LaserStart_Ext()
   LIN {X 1.602, Y -26.386, Z 48.450}
   LaserEnd_Ext()
   LIN {X 1.602, Y -16.134, Z 48.450}
   LaserStart_Ext()
   LIN {X 1.602, Y 38.402, Z 48.450}
   LaserEnd_Ext()
   LIN {X 0.602, Y 40.937, Z 48.450}
   LaserStart_Ext()
   LIN {X 0.602, Y -15.573, Z 48.450}
   LaserEnd_Ext()
   LIN {X 0.602, Y -26.826, Z 48.450}
   LaserStart_Ext()
   LIN {X 0.602, Y -28.931, Z 48.450}
   LaserEnd_Ext()
   LIN {X -0.398, Y -28.998, Z 48.450}
   LaserStart_Ext()
   LIN {X -0.398, Y -27.149, Z 48.450}
   LaserEnd_Ext()
   LIN {X -0.398, Y -15.423, Z 48.450}
   LaserStart_Ext()
   LIN {X -0.398, Y 42.470, Z 48.450}
   LaserEnd_Ext()
   LIN {X -1.398, Y 43.092, Z 48.450}
   LaserStart_Ext()
   LIN {X -1.398, Y 21.242, Z 48.450}
   LaserEnd_Ext()
   LIN {X -1.398, Y 8.634, Z 48.450}
   LaserStart_Ext()
   LIN {X -1.398, Y -15.273, Z 48.450}
   LaserEnd_Ext()
   LIN {X -1.398, Y -27.083, Z 48.450}
   LaserStart_Ext()
   LIN {X -1.398, Y -29.064, Z 48.450}
   LaserEnd_Ext()
   LIN {X -2.398, Y -29.130, Z 48.450}
   LaserStart_Ext()
   LIN {X -2.398, Y -27.004, Z 48.450}
   LaserEnd_Ext()
   LIN {X -2.398, Y -15.450, Z 48.450}
   LaserStart_Ext()
   LIN {X -2.398, Y 0.818, Z 48.450}
   LaserEnd_Ext()
   LIN {X -2.398, Y 29.071, Z 48.450}
   LaserStart_Ext()
   LIN {X -2.398, Y 43.248, Z 48.450}
   LaserEnd_Ext()
   LIN {X -3.398, Y 42.905, Z 48.450}
   LaserStart_Ext()
   LIN {X -3.398, Y 33.459, Z 48.450}
   LaserEnd_Ext()
   LIN {X -3.398, Y -3.781, Z 48.450}
   LaserStart_Ext()
   LIN {X -3.398, Y -15.759, Z 48.450}
   LaserEnd_Ext()
   LIN {X -3.398, Y -26.908, Z 48.450}
   LaserStart_Ext()
   LIN {X -3.398, Y -28.902, Z 48.450}
   LaserEnd_Ext()
   LIN {X -4.398, Y -28.553, Z 48.450}
   LaserStart_Ext()
   LIN {X -4.398, Y -26.328, Z 48.450}
   LaserEnd_Ext()
   LIN {X -4.398, Y -16.083, Z 48.450}
   LaserStart_Ext()
   LIN {X -4.398, Y -7.304, Z 48.450}
   LaserEnd_Ext()
   LIN {X -4.398, Y 36.960, Z 48.450}
   LaserStart_Ext()
   LIN {X -4.398, Y 42.471, Z 48.450}
   LaserEnd_Ext()
   LIN {X -5.398, Y -10.276, Z 48.450}
   LaserStart_Ext()
   LIN {X -5.398, Y -16.962, Z 48.450}
   LaserEnd_Ext()
   LIN {X -5.398, Y -25.687, Z 48.450}
   LaserStart_Ext()
   LIN {X -5.398, Y -28.172, Z 48.450}
   LaserEnd_Ext()
   LIN {X -6.398, Y -27.377, Z 48.450}
   LaserStart_Ext()
   LIN {X -6.398, Y -24.359, Z 48.450}
   LaserEnd_Ext()
   LIN {X -6.398, Y -18.054, Z 48.450}
   LaserStart_Ext()
   LIN {X -6.398, Y -12.872, Z 48.450}
   LaserEnd_Ext()
   LIN {X -7.398, Y -15.265, Z 48.450}
   LaserStart_Ext()
   LIN {X -7.398, Y -26.495, Z 48.450}
   LaserEnd_Ext()
   LIN {X -8.398, Y -24.759, Z 48.450}
   LaserStart_Ext()
   LIN {X -8.398, Y -17.423, Z 48.450}
   LaserEnd_Ext()
   LIN {X 2.262, Y -17.649, Z 49.300}
   LaserStart_Ext()
   LIN {X 3.009, Y -18.928, Z 49.300} C_DIS
   LIN {X 3.541, Y -19.847, Z 49.300} C_DIS
   LIN {X 3.347, Y -21.253, Z 49.300} C_DIS
   LIN {X 3.184, Y -23.345, Z 49.300} C_DIS
   LIN {X 2.974, Y -23.789, Z 49.300} C_DIS
   LIN {X 2.452, Y -24.376, Z 49.300} C_DIS
   LIN {X 1.693, Y -25.189, Z 49.300} C_DIS
   LIN {X -0.009, Y -26.008, Z 49.300} C_DIS
   LIN {X -0.159, Y -26.063, Z 49.300} C_DIS
   LIN {X -0.557, Y -26.032, Z 49.300} C_DIS
   LIN {X -3.064, Y -25.893, Z 49.300} C_DIS
   LIN {X -4.023, Y -25.284, Z 49.300} C_DIS
   LIN {X -4.805, Y -24.782, Z 49.300} C_DIS
   LIN {X -5.510, Y -23.718, Z 49.300} C_DIS
   LIN {X -5.957, Y -23.047, Z 49.300} C_DIS
   LIN {X -6.079, Y -22.298, Z 49.300} C_DIS
   LIN {X -6.288, Y -20.987, Z 49.300} C_DIS
   LIN {X -5.408, Y -18.436, Z 49.300} C_DIS
   LIN {X -5.371, Y -18.328, Z 49.300} C_DIS
   LIN {X -5.297, Y -18.259, Z 49.300} C_DIS
   LIN {X -3.858, Y -16.917, Z 49.300} C_DIS
   LIN {X -2.254, Y -16.421, Z 49.300} C_DIS
   LIN {X -1.568, Y -16.205, Z 49.300} C_DIS
   LIN {X -0.632, Y -16.335, Z 49.300} C_DIS
   LIN {X 0.476, Y -16.499, Z 49.300} C_DIS
   LIN {X 1.222, Y -16.982, Z 49.300} C_DIS
   LIN {X 2.262, Y -17.649, Z 49.300}
   LaserEnd_Ext()
   LIN {X -3.618, Y 29.933, Z 49.300}
   LaserStart_Ext()
   LIN {X -3.768, Y 30.600, Z 49.300} C_DIS
   LIN {X -4.033, Y 31.763, Z 49.300} C_DIS
   LIN {X -4.326, Y 32.892, Z 49.300} C_DIS
   LIN {X -4.626, Y 34.059, Z 49.300} C_DIS
   LIN {X -4.956, Y 35.187, Z 49.300} C_DIS
   LIN {X -5.293, Y 36.334, Z 49.300} C_DIS
   LIN {X -5.530, Y 37.067, Z 49.300} C_DIS
   LIN {X -5.784, Y 37.857, Z 49.300} C_DIS
   LIN {X -5.934, Y 38.301, Z 49.300} C_DIS
   LIN {X -6.186, Y 39.042, Z 49.300} C_DIS
   LIN {X -6.386, Y 40.080, Z 49.300} C_DIS
   LIN {X -6.421, Y 40.281, Z 49.300} C_DIS
   LIN {X -6.386, Y 40.446, Z 49.300} C_DIS
   LIN {X -6.153, Y 41.820, Z 49.300} C_DIS
   LIN {X -5.380, Y 42.995, Z 49.300} C_DIS
   LIN {X -5.200, Y 43.248, Z 49.300} C_DIS
   LIN {X -3.324, Y 44.097, Z 49.300} C_DIS
   LIN {X -2.726, Y 44.346, Z 49.300} C_DIS
   LIN {X -1.507, Y 44.158, Z 49.300} C_DIS
   LIN {X -1.000, Y 44.081, Z 49.300} C_DIS
   LIN {X -0.713, Y 43.890, Z 49.300} C_DIS
   LIN {X 0.446, Y 43.112, Z 49.300} C_DIS
   LIN {X 1.120, Y 42.079, Z 49.300} C_DIS
   LIN {X 1.250, Y 41.879, Z 49.300} C_DIS
   LIN {X 1.365, Y 41.598, Z 49.300} C_DIS
   LIN {X 1.812, Y 40.505, Z 49.300} C_DIS
   LIN {X 2.219, Y 39.470, Z 49.300} C_DIS
   LIN {X 2.513, Y 38.715, Z 49.300} C_DIS
   LIN {X 3.309, Y 36.538, Z 49.300} C_DIS
   LIN {X 3.529, Y 35.941, Z 49.300} C_DIS
   LIN {X 3.597, Y 35.745, Z 49.300} C_DIS
   LIN {X 4.204, Y 33.935, Z 49.300} C_DIS
   LIN {X 4.463, Y 33.166, Z 49.300} C_DIS
   LIN {X 6.304, Y 26.764, Z 49.300} C_DIS
   LIN {X 6.425, Y 26.339, Z 49.300} C_DIS
   LIN {X 6.461, Y 26.185, Z 49.300} C_DIS
   LIN {X 8.299, Y 17.397, Z 49.300} C_DIS
   LIN {X 8.314, Y 17.273, Z 49.300} C_DIS
   LIN {X 9.690, Y 4.539, Z 49.300} C_DIS
   LIN {X 9.718, Y -0.348, Z 49.300} C_DIS
   LIN {X 9.790, Y -2.171, Z 49.300} C_DIS
   LIN {X 9.785, Y -2.450, Z 49.300} C_DIS
   LIN {X 9.543, Y -8.287, Z 49.300} C_DIS
   LIN {X 9.287, Y -11.209, Z 49.300} C_DIS
   LIN {X 9.112, Y -13.056, Z 49.300} C_DIS
   LIN {X 8.803, Y -15.406, Z 49.300} C_DIS
   LIN {X 8.622, Y -16.830, Z 49.300} C_DIS
   LIN {X 8.489, Y -17.677, Z 49.300} C_DIS
   LIN {X 8.151, Y -19.753, Z 49.300} C_DIS
   LIN {X 7.741, Y -21.894, Z 49.300} C_DIS
   LIN {X 7.544, Y -22.959, Z 49.300} C_DIS
   LIN {X 7.131, Y -23.910, Z 49.300} C_DIS
   LIN {X 6.141, Y -26.249, Z 49.300} C_DIS
   LIN {X 4.099, Y -28.357, Z 49.300} C_DIS
   LIN {X 4.008, Y -28.454, Z 49.300} C_DIS
   LIN {X 3.904, Y -28.510, Z 49.300} C_DIS
   LIN {X 0.753, Y -29.933, Z 49.300} C_DIS
   LIN {X -1.715, Y -30.097, Z 49.300} C_DIS
   LIN {X -3.936, Y -29.700, Z 49.300} C_DIS
   LIN {X -5.718, Y -29.078, Z 49.300} C_DIS
   LIN {X -7.369, Y -27.772, Z 49.300} C_DIS
   LIN {X -7.995, Y -27.271, Z 49.300} C_DIS
   LIN {X -9.009, Y -25.510, Z 49.300} C_DIS
   LIN {X -9.870, Y -24.024, Z 49.300} C_DIS
   LIN {X -10.010, Y -22.733, Z 49.300} C_DIS
   LIN {X -10.258, Y -20.334, Z 49.300} C_DIS
   LIN {X -9.744, Y -18.556, Z 49.300} C_DIS
   LIN {X -9.384, Y -17.286, Z 49.300} C_DIS
   LIN {X -8.790, Y -15.996, Z 49.300} C_DIS
   LIN {X -8.070, Y -14.442, Z 49.300} C_DIS
   LIN {X -7.230, Y -12.363, Z 49.300} C_DIS
   LIN {X -6.564, Y -10.713, Z 49.300} C_DIS
   LIN {X -5.423, Y -7.301, Z 49.300} C_DIS
   LIN {X -5.054, Y -6.206, Z 49.300} C_DIS
   LIN {X -4.963, Y -5.867, Z 49.300} C_DIS
   LIN {X -3.889, Y -1.831, Z 49.300} C_DIS
   LIN {X -3.078, Y 2.542, Z 49.300} C_DIS
   LIN {X -2.717, Y 4.439, Z 49.300} C_DIS
   LIN {X -2.362, Y 9.008, Z 49.300} C_DIS
   LIN {X -2.244, Y 10.495, Z 49.300} C_DIS
   LIN {X -2.016, Y 12.649, Z 49.300} C_DIS
   LIN {X -2.228, Y 17.815, Z 49.300} C_DIS
   LIN {X -2.573, Y 23.779, Z 49.300} C_DIS
   LIN {X -2.992, Y 26.561, Z 49.300} C_DIS
   LIN {X -3.109, Y 27.321, Z 49.300} C_DIS
   LIN {X -3.392, Y 28.755, Z 49.300} C_DIS
   LIN {X -3.618, Y 29.933, Z 49.300}
   LaserEnd_Ext()
   LIN {X -0.470, Y 42.522, Z 49.300}
   LaserStart_Ext()
   LIN {X -4.380, Y 42.522, Z 49.300}
   LaserEnd_Ext()
   LIN {X -5.152, Y 41.522, Z 49.300}
   LaserStart_Ext()
   LIN {X 0.290, Y 41.522, Z 49.300}
   LaserEnd_Ext()
   LIN {X 0.725, Y 40.522, Z 49.300}
   LaserStart_Ext()
   LIN {X -5.359, Y 40.522, Z 49.300}
   LaserEnd_Ext()
   LIN {X -5.260, Y 39.522, Z 49.300}
   LaserStart_Ext()
   LIN {X 1.124, Y 39.522, Z 49.300}
   LaserEnd_Ext()
   LIN {X 1.515, Y 38.522, Z 49.300}
   LaserStart_Ext()
   LIN {X -4.953, Y 38.522, Z 49.300}
   LaserEnd_Ext()
   LIN {X -4.626, Y 37.522, Z 49.300}
   LaserStart_Ext()
   LIN {X 1.885, Y 37.522, Z 49.300}
   LaserEnd_Ext()
   LIN {X 2.250, Y 36.522, Z 49.300}
   LaserStart_Ext()
   LIN {X -4.306, Y 36.522, Z 49.300}
   LaserEnd_Ext()
   LIN {X -4.012, Y 35.522, Z 49.300}
   LaserStart_Ext()
   LIN {X 2.616, Y 35.522, Z 49.300}
   LaserEnd_Ext()
   LIN {X 2.953, Y 34.522, Z 49.300}
   LaserStart_Ext()
   LIN {X -3.719, Y 34.522, Z 49.300}
   LaserEnd_Ext()
   LIN {X -3.455, Y 33.522, Z 49.300}
   LaserStart_Ext()
   LIN {X 3.288, Y 33.522, Z 49.300}
   LaserEnd_Ext()
   LIN {X 3.611, Y 32.522, Z 49.300}
   LaserStart_Ext()
   LIN {X -3.197, Y 32.522, Z 49.300}
   LaserEnd_Ext()
   LIN {X -2.953, Y 31.522, Z 49.300}
   LaserStart_Ext()
   LIN {X 3.898, Y 31.522, Z 49.300}
   LaserEnd_Ext()
   LIN {X 4.185, Y 30.522, Z 49.300}
   LaserStart_Ext()
   LIN {X -2.726, Y 30.522, Z 49.300}
   LaserEnd_Ext()
   LIN {X -2.521, Y 29.522, Z 49.300}
   LaserStart_Ext()
   LIN {X 4.472, Y 29.522, Z 49.300}
   LaserEnd_Ext()
   LIN {X 4.759, Y 28.522, Z 49.300}
   LaserStart_Ext()
   LIN {X -2.326, Y 28.522, Z 49.300}
   LaserEnd_Ext()
   LIN {X -2.130, Y 27.522, Z 49.300}
   LaserStart_Ext()
   LIN {X 5.046, Y 27.522, Z 49.300}
   LaserEnd_Ext()
   LIN {X 5.333, Y 26.522, Z 49.300}
   LaserStart_Ext()
   LIN {X -1.975, Y 26.522, Z 49.300}
   LaserEnd_Ext()
   LIN {X -1.824, Y 25.522, Z 49.300}
   LaserStart_Ext()
   LIN {X 5.578, Y 25.522, Z 49.300}
   LaserEnd_Ext()
   LIN {X 5.788, Y 24.522, Z 49.300}
   LaserStart_Ext()
   LIN {X -1.674, Y 24.522, Z 49.300}
   LaserEnd_Ext()
   LIN {X -1.557, Y 23.522, Z 49.300}
   LaserStart_Ext()
   LIN {X 5.997, Y 23.522, Z 49.300}
   LaserEnd_Ext()
   LIN {X 6.206, Y 22.522, Z 49.300}
   LaserStart_Ext()
   LIN {X -1.499, Y 22.522, Z 49.300}
   LaserEnd_Ext()
   LIN {X -1.441, Y 21.522, Z 49.300}
   LaserStart_Ext()
   LIN {X 6.415, Y 21.522, Z 49.300}
   LaserEnd_Ext()
   LIN {X 6.624, Y 20.522, Z 49.300}
   LaserStart_Ext()
   LIN {X -1.383, Y 20.522, Z 49.300}
   LaserEnd_Ext()
   LIN {X -1.325, Y 19.522, Z 49.300}
   LaserStart_Ext()
   LIN {X 6.833, Y 19.522, Z 49.300}
   LaserEnd_Ext()
   LIN {X 7.043, Y 18.522, Z 49.300}
   LaserStart_Ext()
   LIN {X -1.267, Y 18.522, Z 49.300}
   LaserEnd_Ext()
   LIN {X -1.215, Y 17.522, Z 49.300}
   LaserStart_Ext()
   LIN {X 7.252, Y 17.522, Z 49.300}
   LaserEnd_Ext()
   LIN {X 7.390, Y 16.522, Z 49.300}
   LaserStart_Ext()
   LIN {X -1.174, Y 16.522, Z 49.300}
   LaserEnd_Ext()
   LIN {X -1.133, Y 15.522, Z 49.300}
   LaserStart_Ext()
   LIN {X 7.498, Y 15.522, Z 49.300}
   LaserEnd_Ext()
   LIN {X 7.606, Y 14.522, Z 49.300}
   LaserStart_Ext()
   LIN {X -1.092, Y 14.522, Z 49.300}
   LaserEnd_Ext()
   LIN {X -1.051, Y 13.522, Z 49.300}
   LaserStart_Ext()
   LIN {X 7.714, Y 13.522, Z 49.300}
   LaserEnd_Ext()
   LIN {X 7.822, Y 12.522, Z 49.300}
   LaserStart_Ext()
   LIN {X -1.024, Y 12.522, Z 49.300}
   LaserEnd_Ext()
   LIN {X -1.130, Y 11.522, Z 49.300}
   LaserStart_Ext()
   LIN {X 7.930, Y 11.522, Z 49.300}
   LaserEnd_Ext()
   LIN {X 8.038, Y 10.522, Z 49.300}
   LaserStart_Ext()
   LIN {X -1.236, Y 10.522, Z 49.300}
   LaserEnd_Ext()
   LIN {X -1.318, Y 9.522, Z 49.300}
   LaserStart_Ext()
   LIN {X 8.146, Y 9.522, Z 49.300}
   LaserEnd_Ext()
   LIN {X 8.254, Y 8.522, Z 49.300}
   LaserStart_Ext()
   LIN {X -1.397, Y 8.522, Z 49.300}
   LaserEnd_Ext()
   LIN {X -1.475, Y 7.522, Z 49.300}
   LaserStart_Ext()
   LIN {X 8.362, Y 7.522, Z 49.300}
   LaserEnd_Ext()
   LIN {X 8.470, Y 6.522, Z 49.300}
   LaserStart_Ext()
   LIN {X -1.552, Y 6.522, Z 49.300}
   LaserEnd_Ext()
   LIN {X -1.630, Y 5.522, Z 49.300}
   LaserStart_Ext()
   LIN {X 8.578, Y 5.522, Z 49.300}
   LaserEnd_Ext()
   LIN {X 8.686, Y 4.522, Z 49.300}
   LaserStart_Ext()
   LIN {X -1.708, Y 4.522, Z 49.300}
   LaserEnd_Ext()
   LIN {X -1.874, Y 3.522, Z 49.300}
   LaserStart_Ext()
   LIN {X 8.696, Y 3.522, Z 49.300}
   LaserEnd_Ext()
   LIN {X 8.702, Y 2.522, Z 49.300}
   LaserStart_Ext()
   LIN {X -2.064, Y 2.522, Z 49.300}
   LaserEnd_Ext()
   LIN {X -2.251, Y 1.522, Z 49.300}
   LaserStart_Ext()
   LIN {X 8.707, Y 1.522, Z 49.300}
   LaserEnd_Ext()
   LIN {X 8.713, Y 0.522, Z 49.300}
   LaserStart_Ext()
   LIN {X -2.436, Y 0.522, Z 49.300}
   LaserEnd_Ext()
   LIN {X -2.621, Y -0.478, Z 49.300}
   LaserStart_Ext()
   LIN {X 8.723, Y -0.478, Z 49.300}
   LaserEnd_Ext()
   LIN {X 8.762, Y -1.478, Z 49.300}
   LaserStart_Ext()
   LIN {X -2.807, Y -1.478, Z 49.300}
   LaserEnd_Ext()
   LIN {X -3.026, Y -2.478, Z 49.300}
   LaserStart_Ext()
   LIN {X 8.783, Y -2.478, Z 49.300}
   LaserEnd_Ext()
   LIN {X 8.742, Y -3.478, Z 49.300}
   LaserStart_Ext()
   LIN {X -3.293, Y -3.478, Z 49.300}
   LaserEnd_Ext()
   LIN {X -3.559, Y -4.478, Z 49.300}
   LaserStart_Ext()
   LIN {X 8.700, Y -4.478, Z 49.300}
   LaserEnd_Ext()
   LIN {X 8.659, Y -5.478, Z 49.300}
   LaserStart_Ext()
   LIN {X -3.825, Y -5.478, Z 49.300}
   LaserEnd_Ext()
   LIN {X -4.092, Y -6.478, Z 49.300}
   LaserStart_Ext()
   LIN {X 8.617, Y -6.478, Z 49.300}
   LaserEnd_Ext()
   LIN {X 8.576, Y -7.478, Z 49.300}
   LaserStart_Ext()
   LIN {X -4.427, Y -7.478, Z 49.300}
   LaserEnd_Ext()
   LIN {X -4.762, Y -8.478, Z 49.300}
   LaserStart_Ext()
   LIN {X 8.523, Y -8.478, Z 49.300}
   LaserEnd_Ext()
   LIN {X 8.435, Y -9.478, Z 49.300}
   LaserStart_Ext()
   LIN {X -5.097, Y -9.478, Z 49.300}
   LaserEnd_Ext()
   LIN {X -5.431, Y -10.478, Z 49.300}
   LaserStart_Ext()
   LIN {X 8.347, Y -10.478, Z 49.300}
   LaserEnd_Ext()
   LIN {X 8.257, Y -11.478, Z 49.300}
   LaserStart_Ext()
   LIN {X -5.795, Y -11.478, Z 49.300}
   LaserEnd_Ext()
   LIN {X -6.198, Y -12.478, Z 49.300}
   LaserStart_Ext()
   LIN {X 8.162, Y -12.478, Z 49.300}
   LaserEnd_Ext()
   LIN {X 8.048, Y -13.478, Z 49.300}
   LaserStart_Ext()
   LIN {X -6.602, Y -13.478, Z 49.300}
   LaserEnd_Ext()
   LIN {X -7.006, Y -14.478, Z 49.300}
   LaserStart_Ext()
   LIN {X 7.917, Y -14.478, Z 49.300}
   LaserEnd_Ext()
   LIN {X 7.786, Y -15.478, Z 49.300}
   LaserStart_Ext()
   LIN {X 0.411, Y -15.478, Z 49.300}
   LaserEnd_Ext()
   LIN {X -2.589, Y -15.478, Z 49.300}
   LaserStart_Ext()
   LIN {X -7.448, Y -15.478, Z 49.300}
   LaserEnd_Ext()
   LIN {X -7.911, Y -16.478, Z 49.300}
   LaserStart_Ext()
   LIN {X -4.854, Y -16.478, Z 49.300}
   LaserEnd_Ext()
   LIN {X 2.290, Y -16.478, Z 49.300}
   LaserStart_Ext()
   LIN {X 7.659, Y -16.478, Z 49.300}
   LaserEnd_Ext()
   LIN {X 7.508, Y -17.478, Z 49.300}
   LaserStart_Ext()
   LIN {X 3.321, Y -17.478, Z 49.300}
   LaserEnd_Ext()
   LIN {X -5.926, Y -17.478, Z 49.300}
   LaserStart_Ext()
   LIN {X -8.371, Y -17.478, Z 49.300}
   LaserEnd_Ext()
   LIN {X -8.683, Y -18.478, Z 49.300}
   LaserStart_Ext()
   LIN {X -6.480, Y -18.478, Z 49.300}
   LaserEnd_Ext()
   LIN {X 3.904, Y -18.478, Z 49.300}
   LaserStart_Ext()
   LIN {X 7.345, Y -18.478, Z 49.300}
   LaserEnd_Ext()
   LIN {X 7.183, Y -19.478, Z 49.300}
   LaserStart_Ext()
   LIN {X 4.470, Y -19.478, Z 49.300}
   LaserEnd_Ext()
   LIN {X -6.825, Y -19.478, Z 49.300}
   LaserStart_Ext()
   LIN {X -8.970, Y -19.478, Z 49.300}
   LaserEnd_Ext()
   LIN {X -9.238, Y -20.478, Z 49.300}
   LaserStart_Ext()
   LIN {X -7.171, Y -20.478, Z 49.300}
   LaserEnd_Ext()
   LIN {X 4.464, Y -20.478, Z 49.300}
   LaserStart_Ext()
   LIN {X 6.994, Y -20.478, Z 49.300}
   LaserEnd_Ext()
   LIN {X 6.802, Y -21.478, Z 49.300}
   LaserStart_Ext()
   LIN {X 4.333, Y -21.478, Z 49.300}
   LaserEnd_Ext()
   LIN {X -7.222, Y -21.478, Z 49.300}
   LaserStart_Ext()
   LIN {X -9.134, Y -21.478, Z 49.300}
   LaserEnd_Ext()
   LIN {X -9.031, Y -22.478, Z 49.300}
   LaserStart_Ext()
   LIN {X -7.063, Y -22.478, Z 49.300}
   LaserEnd_Ext()
   LIN {X 4.254, Y -22.478, Z 49.300}
   LaserStart_Ext()
   LIN {X 6.616, Y -22.478, Z 49.300}
   LaserEnd_Ext()
   LIN {X 6.228, Y -23.478, Z 49.300}
   LaserStart_Ext()
   LIN {X 4.174, Y -23.478, Z 49.300}
   LaserEnd_Ext()
   LIN {X -6.858, Y -23.478, Z 49.300}
   LaserStart_Ext()
   LIN {X -8.923, Y -23.478, Z 49.300}
   LaserEnd_Ext()
   LIN {X -8.451, Y -24.478, Z 49.300}
   LaserStart_Ext()
   LIN {X -6.206, Y -24.478, Z 49.300}
   LaserEnd_Ext()
   LIN {X 3.699, Y -24.478, Z 49.300}
   LaserStart_Ext()
   LIN {X 5.804, Y -24.478, Z 49.300}
   LaserEnd_Ext()
   LIN {X 5.381, Y -25.478, Z 49.300}
   LaserStart_Ext()
   LIN {X 2.791, Y -25.478, Z 49.300}
   LaserEnd_Ext()
   LIN {X -5.522, Y -25.478, Z 49.300}
   LaserStart_Ext()
   LIN {X -7.873, Y -25.478, Z 49.300}
   LaserEnd_Ext()
   LIN {X -7.297, Y -26.478, Z 49.300}
   LaserStart_Ext()
   LIN {X -4.008, Y -26.478, Z 49.300}
   LaserEnd_Ext()
   LIN {X 1.320, Y -26.478, Z 49.300}
   LaserStart_Ext()
   LIN {X 4.526, Y -26.478, Z 49.300}
   LaserEnd_Ext()
   LIN {X 3.558, Y -27.478, Z 49.300}
   LaserStart_Ext()
   LIN {X -6.129, Y -27.478, Z 49.300}
   LaserEnd_Ext()
   LIN {X -4.402, Y -28.478, Z 49.300}
   LaserStart_Ext()
   LIN {X 1.544, Y -28.478, Z 49.300}
   LaserEnd_Ext()
   LIN {X 0.983, Y -16.725, Z 50.150}
   LaserStart_Ext()
   LIN {X 2.331, Y -17.590, Z 50.150} C_DIS
   LIN {X 3.296, Y -19.243, Z 50.150} C_DIS
   LIN {X 3.615, Y -19.785, Z 50.150} C_DIS
   LIN {X 3.605, Y -20.490, Z 50.150} C_DIS
   LIN {X 3.412, Y -22.958, Z 50.150} C_DIS
   LIN {X 3.020, Y -23.788, Z 50.150} C_DIS
   LIN {X 2.042, Y -24.888, Z 50.150} C_DIS
   LIN {X 1.888, Y -25.053, Z 50.150} C_DIS
   LIN {X 1.459, Y -25.259, Z 50.150} C_DIS
   LIN {X -0.277, Y -26.042, Z 50.150} C_DIS
   LIN {X -1.372, Y -25.935, Z 50.150} C_DIS
   LIN {X -2.975, Y -25.847, Z 50.150} C_DIS
   LIN {X -4.420, Y -24.929, Z 50.150} C_DIS
   LIN {X -4.720, Y -24.740, Z 50.150} C_DIS
   LIN {X -4.875, Y -24.509, Z 50.150} C_DIS
   LIN {X -5.875, Y -23.007, Z 50.150} C_DIS
   LIN {X -6.183, Y -21.119, Z 50.150} C_DIS
   LIN {X -6.211, Y -20.948, Z 50.150} C_DIS
   LIN {X -6.156, Y -20.786, Z 50.150} C_DIS
   LIN {X -5.288, Y -18.271, Z 50.150} C_DIS
   LIN {X -4.039, Y -17.112, Z 50.150} C_DIS
   LIN {X -3.766, Y -16.858, Z 50.150} C_DIS
   LIN {X -3.498, Y -16.775, Z 50.150} C_DIS
   LIN {X -1.546, Y -16.158, Z 50.150} C_DIS
   LIN {X 0.096, Y -16.387, Z 50.150} C_DIS
   LIN {X 0.542, Y -16.444, Z 50.150} C_DIS
   LIN {X 0.983, Y -16.725, Z 50.150}
   LaserEnd_Ext()
   LIN {X -6.488, Y 40.328, Z 50.150}
   LaserStart_Ext()
   LIN {X -6.298, Y 41.538, Z 50.150} C_DIS
   LIN {X -6.263, Y 41.758, Z 50.150} C_DIS
   LIN {X -6.147, Y 41.936, Z 50.150} C_DIS
   LIN {X -5.277, Y 43.286, Z 50.150} C_DIS
   LIN {X -2.802, Y 44.392, Z 50.150} C_DIS
   LIN {X -2.231, Y 44.307, Z 50.150} C_DIS
   LIN {X -1.076, Y 44.132, Z 50.150} C_DIS
   LIN {X 0.319, Y 43.201, Z 50.150} C_DIS
   LIN {X 0.396, Y 43.130, Z 50.150} C_DIS
   LIN {X 1.180, Y 41.935, Z 50.150} C_DIS
   LIN {X 1.600, Y 40.917, Z 50.150} C_DIS
   LIN {X 1.745, Y 40.563, Z 50.150} C_DIS
   LIN {X 2.001, Y 39.912, Z 50.150} C_DIS
   LIN {X 2.428, Y 38.830, Z 50.150} C_DIS
   LIN {X 2.819, Y 37.786, Z 50.150} C_DIS
   LIN {X 3.357, Y 36.325, Z 50.150} C_DIS
   LIN {X 3.884, Y 34.807, Z 50.150} C_DIS
   LIN {X 4.406, Y 33.250, Z 50.150} C_DIS
   LIN {X 5.654, Y 28.901, Z 50.150} C_DIS
   LIN {X 6.219, Y 26.985, Z 50.150} C_DIS
   LIN {X 6.467, Y 26.115, Z 50.150} C_DIS
   LIN {X 8.132, Y 18.164, Z 50.150} C_DIS
   LIN {X 8.400, Y 16.756, Z 50.150} C_DIS
   LIN {X 8.505, Y 15.674, Z 50.150} C_DIS
   LIN {X 9.713, Y 4.493, Z 50.150} C_DIS
   LIN {X 9.737, Y 0.263, Z 50.150} C_DIS
   LIN {X 9.799, Y -1.314, Z 50.150} C_DIS
   LIN {X 9.825, Y -2.050, Z 50.150} C_DIS
   LIN {X 9.743, Y -4.534, Z 50.150} C_DIS
   LIN {X 9.590, Y -8.211, Z 50.150} C_DIS
   LIN {X 9.191, Y -12.767, Z 50.150} C_DIS
   LIN {X 9.170, Y -12.981, Z 50.150} C_DIS
   LIN {X 9.135, Y -13.253, Z 50.150} C_DIS
   LIN {X 8.689, Y -16.756, Z 50.150} C_DIS
   LIN {X 8.362, Y -18.839, Z 50.150} C_DIS
   LIN {X 8.225, Y -19.681, Z 50.150} C_DIS
   LIN {X 8.059, Y -20.549, Z 50.150} C_DIS
   LIN {X 7.625, Y -22.888, Z 50.150} C_DIS
   LIN {X 6.720, Y -24.976, Z 50.150} C_DIS
   LIN {X 6.176, Y -26.260, Z 50.150} C_DIS
   LIN {X 4.950, Y -27.525, Z 50.150} C_DIS
   LIN {X 3.954, Y -28.492, Z 50.150} C_DIS
   LIN {X 2.399, Y -29.111, Z 50.150} C_DIS
   LIN {X 0.523, Y -29.957, Z 50.150} C_DIS
   LIN {X -0.828, Y -30.047, Z 50.150} C_DIS
   LIN {X -4.726, Y -29.351, Z 50.150} C_DIS
   LIN {X -5.623, Y -29.038, Z 50.150} C_DIS
   LIN {X -7.464, Y -27.582, Z 50.150} C_DIS
   LIN {X -7.903, Y -27.236, Z 50.150} C_DIS
   LIN {X -8.079, Y -26.938, Z 50.150} C_DIS
   LIN {X -9.786, Y -23.994, Z 50.150} C_DIS
   LIN {X -10.143, Y -20.691, Z 50.150} C_DIS
   LIN {X -10.183, Y -20.305, Z 50.150} C_DIS
   LIN {X -10.100, Y -20.018, Z 50.150} C_DIS
   LIN {X -9.316, Y -17.255, Z 50.150} C_DIS
   LIN {X -8.123, Y -14.665, Z 50.150} C_DIS
   LIN {X -8.079, Y -14.568, Z 50.150} C_DIS
   LIN {X -8.021, Y -14.421, Z 50.150} C_DIS
   LIN {X -6.531, Y -10.728, Z 50.150} C_DIS
   LIN {X -5.452, Y -7.503, Z 50.150} C_DIS
   LIN {X -5.063, Y -6.338, Z 50.150} C_DIS
   LIN {X -4.791, Y -5.313, Z 50.150} C_DIS
   LIN {X -3.890, Y -1.930, Z 50.150} C_DIS
   LIN {X -2.791, Y 4.000, Z 50.150} C_DIS
   LIN {X -2.705, Y 4.453, Z 50.150} C_DIS
   LIN {X -2.280, Y 9.927, Z 50.150} C_DIS
   LIN {X -2.192, Y 11.040, Z 50.150} C_DIS
   LIN {X -2.021, Y 12.652, Z 50.150} C_DIS
   LIN {X -2.179, Y 16.519, Z 50.150} C_DIS
   LIN {X -2.604, Y 23.843, Z 50.150} C_DIS
   LIN {X -3.059, Y 26.868, Z 50.150} C_DIS
   LIN {X -3.134, Y 27.287, Z 50.150} C_DIS
   LIN {X -3.558, Y 29.492, Z 50.150} C_DIS
   LIN {X -3.982, Y 31.377, Z 50.150} C_DIS
   LIN {X -4.080, Y 31.806, Z 50.150} C_DIS
   LIN {X -4.366, Y 32.910, Z 50.150} C_DIS
   LIN {X -4.678, Y 34.101, Z 50.150} C_DIS
   LIN {X -5.139, Y 35.657, Z 50.150} C_DIS
   LIN {X -5.350, Y 36.375, Z 50.150} C_DIS
   LIN {X -5.512, Y 36.874, Z 50.150} C_DIS
   LIN {X -5.845, Y 37.897, Z 50.150} C_DIS
   LIN {X -6.177, Y 38.865, Z 50.150} C_DIS
   LIN {X -6.250, Y 39.081, Z 50.150} C_DIS
   LIN {X -6.281, Y 39.241, Z 50.150} C_DIS
   LIN {X -6.488, Y 40.328, Z 50.150}
   LaserEnd_Ext()
   LIN {X -8.280, Y -17.396, Z 50.150}
   LaserStart_Ext()
   LIN {X -8.280, Y -24.598, Z 50.150}
   LaserEnd_Ext()
   LIN {X -7.280, Y -26.322, Z 50.150}
   LaserStart_Ext()
   LIN {X -7.280, Y -15.224, Z 50.150}
   LaserEnd_Ext()
   LIN {X -6.280, Y -12.778, Z 50.150}
   LaserStart_Ext()
   LIN {X -6.280, Y -18.079, Z 50.150}
   LaserEnd_Ext()
   LIN {X -6.280, Y -24.204, Z 50.150}
   LaserStart_Ext()
   LIN {X -6.280, Y -27.243, Z 50.150}
   LaserEnd_Ext()
   LIN {X -5.280, Y -28.035, Z 50.150}
   LaserStart_Ext()
   LIN {X -5.280, Y -25.567, Z 50.150}
   LaserEnd_Ext()
   LIN {X -5.280, Y -16.899, Z 50.150}
   LaserStart_Ext()
   LIN {X -5.280, Y -10.140, Z 50.150}
   LaserEnd_Ext()
   LIN {X -5.280, Y 39.334, Z 50.150}
   LaserStart_Ext()
   LIN {X -5.280, Y 41.436, Z 50.150}
   LaserEnd_Ext()
   LIN {X -4.280, Y 42.636, Z 50.150}
   LaserStart_Ext()
   LIN {X -4.280, Y 36.279, Z 50.150}
   LaserEnd_Ext()
   LIN {X -4.280, Y -7.150, Z 50.150}
   LaserStart_Ext()
   LIN {X -4.280, Y -16.001, Z 50.150}
   LaserEnd_Ext()
   LIN {X -4.280, Y -26.203, Z 50.150}
   LaserStart_Ext()
   LIN {X -4.280, Y -28.415, Z 50.150}
   LaserEnd_Ext()
   LIN {X -3.280, Y -28.594, Z 50.150}
   LaserStart_Ext()
   LIN {X -3.280, Y -26.798, Z 50.150}
   LaserEnd_Ext()
   LIN {X -3.280, Y -15.657, Z 50.150}
   LaserStart_Ext()
   LIN {X -3.280, Y -3.525, Z 50.150}
   LaserEnd_Ext()
   LIN {X -3.280, Y 32.704, Z 50.150}
   LaserStart_Ext()
   LIN {X -3.280, Y 43.084, Z 50.150}
   LaserEnd_Ext()
   LIN {X -2.280, Y 43.303, Z 50.150}
   LaserStart_Ext()
   LIN {X -2.280, Y 28.141, Z 50.150}
   LaserEnd_Ext()
   LIN {X -2.280, Y 1.272, Z 50.150}
   LaserStart_Ext()
   LIN {X -2.280, Y -15.341, Z 50.150}
   LaserEnd_Ext()
   LIN {X -2.280, Y -26.887, Z 50.150}
   LaserStart_Ext()
   LIN {X -2.280, Y -28.772, Z 50.150}
   LaserEnd_Ext()
   LIN {X -1.280, Y -28.951, Z 50.150}
   LaserStart_Ext()
   LIN {X -1.280, Y -26.949, Z 50.150}
   LaserEnd_Ext()
   LIN {X -1.280, Y -15.186, Z 50.150}
   LaserStart_Ext()
   LIN {X -1.280, Y 9.887, Z 50.150}
   LaserEnd_Ext()
   LIN {X -1.280, Y 18.283, Z 50.150}
   LaserStart_Ext()
   LIN {X -1.280, Y 43.066, Z 50.150}
   LaserEnd_Ext()
   LIN {X -0.280, Y 42.337, Z 50.150}
   LaserStart_Ext()
   LIN {X -0.280, Y -15.325, Z 50.150}
   LaserEnd_Ext()
   LIN {X -0.280, Y -27.042, Z 50.150}
   LaserStart_Ext()
   LIN {X -0.280, Y -29.009, Z 50.150}
   LaserEnd_Ext()
   LIN {X 0.720, Y -28.771, Z 50.150}
   LaserStart_Ext()
   LIN {X 0.720, Y -26.689, Z 50.150}
   LaserEnd_Ext()
   LIN {X 0.720, Y -15.462, Z 50.150}
   LaserStart_Ext()
   LIN {X 0.720, Y 40.426, Z 50.150}
   LaserEnd_Ext()
   LIN {X 1.720, Y 37.869, Z 50.150}
   LaserStart_Ext()
   LIN {X 1.720, Y -16.010, Z 50.150}
   LaserEnd_Ext()
   LIN {X 1.720, Y -26.238, Z 50.150}
   LaserStart_Ext()
   LIN {X 1.720, Y -28.320, Z 50.150}
   LaserEnd_Ext()
   LIN {X 2.720, Y -27.906, Z 50.150}
   LaserStart_Ext()
   LIN {X 2.720, Y -25.627, Z 50.150}
   LaserEnd_Ext()
   LIN {X 2.720, Y -16.651, Z 50.150}
   LaserStart_Ext()
   LIN {X 2.720, Y 35.110, Z 50.150}
   LaserEnd_Ext()
   LIN {X 3.720, Y 32.016, Z 50.150}
   LaserStart_Ext()
   LIN {X 3.720, Y -17.985, Z 50.150}
   LaserEnd_Ext()
   LIN {X 3.720, Y -24.506, Z 50.150}
   LaserStart_Ext()
   LIN {X 3.720, Y -27.325, Z 50.150}
   LaserEnd_Ext()
   LIN {X 4.720, Y -26.325, Z 50.150}
   LaserStart_Ext()
   LIN {X 4.720, Y 28.533, Z 50.150}
   LaserEnd_Ext()
   LIN {X 5.720, Y 24.801, Z 50.150}
   LaserStart_Ext()
   LIN {X 5.720, Y -24.771, Z 50.150}
   LaserEnd_Ext()
   LIN {X 6.720, Y -22.284, Z 50.150}
   LaserStart_Ext()
   LIN {X 6.720, Y 20.026, Z 50.150}
   LaserEnd_Ext()
   LIN {X 7.720, Y 13.625, Z 50.150}
   LaserStart_Ext()
   LIN {X 7.720, Y -16.451, Z 50.150}
   LaserEnd_Ext()
   LIN {X 8.720, Y -5.056, Z 50.150}
   LaserStart_Ext()
   LIN {X 8.720, Y 3.197, Z 50.150}
   LaserEnd_Ext()
   LIN {X -1.136, Y -16.166, Z 51.000}
   LaserStart_Ext()
   LIN {X 0.608, Y -16.390, Z 51.000} C_DIS
   LIN {X 2.334, Y -17.488, Z 51.000} C_DIS
   LIN {X 2.448, Y -17.613, Z 51.000} C_DIS
   LIN {X 3.690, Y -19.723, Z 51.000} C_DIS
   LIN {X 3.648, Y -22.468, Z 51.000} C_DIS
   LIN {X 3.640, Y -22.570, Z 51.000} C_DIS
   LIN {X 3.066, Y -23.787, Z 51.000} C_DIS
   LIN {X 2.371, Y -24.569, Z 51.000} C_DIS
   LIN {X 1.821, Y -25.099, Z 51.000} C_DIS
   LIN {X 0.911, Y -25.408, Z 51.000} C_DIS
   LIN {X -0.481, Y -26.035, Z 51.000} C_DIS
   LIN {X -2.880, Y -25.802, Z 51.000} C_DIS
   LIN {X -4.634, Y -24.698, Z 51.000} C_DIS
   LIN {X -5.541, Y -23.348, Z 51.000} C_DIS
   LIN {X -5.794, Y -22.968, Z 51.000} C_DIS
   LIN {X -5.872, Y -22.491, Z 51.000} C_DIS
   LIN {X -6.134, Y -20.909, Z 51.000} C_DIS
   LIN {X -5.621, Y -19.416, Z 51.000} C_DIS
   LIN {X -5.206, Y -18.214, Z 51.000} C_DIS
   LIN {X -4.393, Y -17.460, Z 51.000} C_DIS
   LIN {X -3.674, Y -16.798, Z 51.000} C_DIS
   LIN {X -2.139, Y -16.306, Z 51.000} C_DIS
   LIN {X -1.523, Y -16.112, Z 51.000} C_DIS
   LIN {X -1.136, Y -16.166, Z 51.000}
   LaserEnd_Ext()
   LIN {X -7.227, Y -12.550, Z 51.000}
   LaserStart_Ext()
   LIN {X -6.498, Y -10.744, Z 51.000} C_DIS
   LIN {X -5.970, Y -9.167, Z 51.000} C_DIS
   LIN {X -5.082, Y -6.505, Z 51.000} C_DIS
   LIN {X -4.459, Y -4.162, Z 51.000} C_DIS
   LIN {X -3.892, Y -2.029, Z 51.000} C_DIS
   LIN {X -3.043, Y 2.549, Z 51.000} C_DIS
   LIN {X -2.757, Y 4.062, Z 51.000} C_DIS
   LIN {X -2.683, Y 4.546, Z 51.000} C_DIS
   LIN {X -2.530, Y 6.571, Z 51.000} C_DIS
   LIN {X -2.198, Y 10.846, Z 51.000} C_DIS
   LIN {X -2.139, Y 11.585, Z 51.000} C_DIS
   LIN {X -2.026, Y 12.655, Z 51.000} C_DIS
   LIN {X -2.131, Y 15.223, Z 51.000} C_DIS
   LIN {X -2.634, Y 23.906, Z 51.000} C_DIS
   LIN {X -3.008, Y 26.394, Z 51.000} C_DIS
   LIN {X -3.310, Y 28.073, Z 51.000} C_DIS
   LIN {X -3.498, Y 29.052, Z 51.000} C_DIS
   LIN {X -3.883, Y 30.763, Z 51.000} C_DIS
   LIN {X -4.127, Y 31.850, Z 51.000} C_DIS
   LIN {X -4.474, Y 33.163, Z 51.000} C_DIS
   LIN {X -4.730, Y 34.143, Z 51.000} C_DIS
   LIN {X -4.935, Y 34.833, Z 51.000} C_DIS
   LIN {X -5.408, Y 36.415, Z 51.000} C_DIS
   LIN {X -5.863, Y 37.804, Z 51.000} C_DIS
   LIN {X -5.906, Y 37.936, Z 51.000} C_DIS
   LIN {X -6.314, Y 39.119, Z 51.000} C_DIS
   LIN {X -6.517, Y 40.189, Z 51.000} C_DIS
   LIN {X -6.555, Y 40.393, Z 51.000} C_DIS
   LIN {X -6.519, Y 40.617, Z 51.000} C_DIS
   LIN {X -6.326, Y 41.815, Z 51.000} C_DIS
   LIN {X -5.469, Y 43.135, Z 51.000} C_DIS
   LIN {X -5.337, Y 43.340, Z 51.000} C_DIS
   LIN {X -2.878, Y 44.439, Z 51.000} C_DIS
   LIN {X -1.508, Y 44.235, Z 51.000} C_DIS
   LIN {X -1.152, Y 44.182, Z 51.000} C_DIS
   LIN {X -0.979, Y 44.069, Z 51.000} C_DIS
   LIN {X 0.299, Y 43.220, Z 51.000} C_DIS
   LIN {X 1.057, Y 42.070, Z 51.000} C_DIS
   LIN {X 1.160, Y 41.867, Z 51.000} C_DIS
   LIN {X 1.678, Y 40.620, Z 51.000} C_DIS
   LIN {X 2.056, Y 39.673, Z 51.000} C_DIS
   LIN {X 2.325, Y 38.990, Z 51.000} C_DIS
   LIN {X 2.825, Y 37.657, Z 51.000} C_DIS
   LIN {X 3.184, Y 36.707, Z 51.000} C_DIS
   LIN {X 3.298, Y 36.393, Z 51.000} C_DIS
   LIN {X 3.745, Y 35.096, Z 51.000} C_DIS
   LIN {X 4.171, Y 33.869, Z 51.000} C_DIS
   LIN {X 4.321, Y 33.421, Z 51.000} C_DIS
   LIN {X 4.680, Y 32.169, Z 51.000} C_DIS
   LIN {X 5.943, Y 27.881, Z 51.000} C_DIS
   LIN {X 6.499, Y 25.932, Z 51.000} C_DIS
   LIN {X 7.947, Y 19.015, Z 51.000} C_DIS
   LIN {X 8.500, Y 16.115, Z 51.000} C_DIS
   LIN {X 8.715, Y 13.887, Z 51.000} C_DIS
   LIN {X 9.735, Y 4.446, Z 51.000} C_DIS
   LIN {X 9.756, Y 0.875, Z 51.000} C_DIS
   LIN {X 9.808, Y -0.456, Z 51.000} C_DIS
   LIN {X 9.858, Y -1.865, Z 51.000} C_DIS
   LIN {X 9.700, Y -6.618, Z 51.000} C_DIS
   LIN {X 9.638, Y -8.135, Z 51.000} C_DIS
   LIN {X 9.450, Y -10.267, Z 51.000} C_DIS
   LIN {X 9.229, Y -12.906, Z 51.000} C_DIS
   LIN {X 9.096, Y -14.014, Z 51.000} C_DIS
   LIN {X 8.757, Y -16.682, Z 51.000} C_DIS
   LIN {X 8.357, Y -19.221, Z 51.000} C_DIS
   LIN {X 8.299, Y -19.608, Z 51.000} C_DIS
   LIN {X 8.231, Y -19.987, Z 51.000} C_DIS
   LIN {X 7.707, Y -22.816, Z 51.000} C_DIS
   LIN {X 6.308, Y -26.041, Z 51.000} C_DIS
   LIN {X 6.211, Y -26.271, Z 51.000} C_DIS
   LIN {X 5.992, Y -26.497, Z 51.000} C_DIS
   LIN {X 3.895, Y -28.532, Z 51.000} C_DIS
   LIN {X 0.620, Y -29.835, Z 51.000} C_DIS
   LIN {X 0.294, Y -29.982, Z 51.000} C_DIS
   LIN {X 0.059, Y -29.998, Z 51.000} C_DIS
   LIN {X -5.517, Y -29.002, Z 51.000} C_DIS
   LIN {X -7.812, Y -27.201, Z 51.000} C_DIS
   LIN {X -8.716, Y -25.665, Z 51.000} C_DIS
   LIN {X -9.703, Y -23.963, Z 51.000} C_DIS
   LIN {X -9.953, Y -21.644, Z 51.000} C_DIS
   LIN {X -10.107, Y -20.275, Z 51.000} C_DIS
   LIN {X -9.758, Y -19.023, Z 51.000} C_DIS
   LIN {X -9.248, Y -17.223, Z 51.000} C_DIS
   LIN {X -8.607, Y -15.831, Z 51.000} C_DIS
   LIN {X -8.018, Y -14.536, Z 51.000} C_DIS
   LIN {X -7.227, Y -12.550, Z 51.000}
   LaserEnd_Ext()
   LIN {X 1.621, Y -28.360, Z 51.000}
   LaserStart_Ext()
   LIN {X -3.423, Y -28.360, Z 51.000}
   LaserEnd_Ext()
   LIN {X -5.992, Y -27.360, Z 51.000}
   LaserStart_Ext()
   LIN {X 3.666, Y -27.360, Z 51.000}
   LaserEnd_Ext()
   LIN {X 4.697, Y -26.360, Z 51.000}
   LaserStart_Ext()
   LIN {X 1.231, Y -26.360, Z 51.000}
   LaserEnd_Ext()
   LIN {X -3.874, Y -26.360, Z 51.000}
   LaserStart_Ext()
   LIN {X -7.146, Y -26.360, Z 51.000}
   LaserEnd_Ext()
   LIN {X -7.735, Y -25.360, Z 51.000}
   LaserStart_Ext()
   LIN {X -5.381, Y -25.360, Z 51.000}
   LaserEnd_Ext()
   LIN {X 2.991, Y -25.360, Z 51.000}
   LaserStart_Ext()
   LIN {X 5.513, Y -25.360, Z 51.000}
   LaserEnd_Ext()
   LIN {X 5.947, Y -24.360, Z 51.000}
   LaserStart_Ext()
   LIN {X 3.885, Y -24.360, Z 51.000}
   LaserEnd_Ext()
   LIN {X -6.065, Y -24.360, Z 51.000}
   LaserStart_Ext()
   LIN {X -8.316, Y -24.360, Z 51.000}
   LaserEnd_Ext()
   LIN {X -8.762, Y -23.360, Z 51.000}
   LaserStart_Ext()
   LIN {X -6.712, Y -23.360, Z 51.000}
   LaserEnd_Ext()
   LIN {X 4.373, Y -23.360, Z 51.000}
   LaserStart_Ext()
   LIN {X 6.381, Y -23.360, Z 51.000}
   LaserEnd_Ext()
   LIN {X 6.774, Y -22.360, Z 51.000}
   LaserStart_Ext()
   LIN {X 4.650, Y -22.360, Z 51.000}
   LaserEnd_Ext()
   LIN {X -6.907, Y -22.360, Z 51.000}
   LaserStart_Ext()
   LIN {X -8.870, Y -22.360, Z 51.000}
   LaserEnd_Ext()
   LIN {X -8.979, Y -21.360, Z 51.000}
   LaserStart_Ext()
   LIN {X -7.073, Y -21.360, Z 51.000}
   LaserEnd_Ext()
   LIN {X 4.665, Y -21.360, Z 51.000}
   LaserStart_Ext()
   LIN {X 6.960, Y -21.360, Z 51.000}
   LaserEnd_Ext()
   LIN {X 7.145, Y -20.360, Z 51.000}
   LaserStart_Ext()
   LIN {X 4.680, Y -20.360, Z 51.000}
   LaserEnd_Ext()
   LIN {X -7.003, Y -20.360, Z 51.000}
   LaserStart_Ext()
   LIN {X -9.092, Y -20.360, Z 51.000}
   LaserEnd_Ext()
   LIN {X -8.814, Y -19.360, Z 51.000}
   LaserStart_Ext()
   LIN {X -6.659, Y -19.360, Z 51.000}
   LaserEnd_Ext()
   LIN {X 4.621, Y -19.360, Z 51.000}
   LaserStart_Ext()
   LIN {X 7.325, Y -19.360, Z 51.000}
   LaserEnd_Ext()
   LIN {X 7.481, Y -18.360, Z 51.000}
   LaserStart_Ext()
   LIN {X 4.048, Y -18.360, Z 51.000}
   LaserEnd_Ext()
   LIN {X -6.314, Y -18.360, Z 51.000}
   LaserStart_Ext()
   LIN {X -8.531, Y -18.360, Z 51.000}
   LaserEnd_Ext()
   LIN {X -8.210, Y -17.360, Z 51.000}
   LaserStart_Ext()
   LIN {X -5.756, Y -17.360, Z 51.000}
   LaserEnd_Ext()
   LIN {X 3.460, Y -17.360, Z 51.000}
   LaserStart_Ext()
   LIN {X 7.638, Y -17.360, Z 51.000}
   LaserEnd_Ext()
   LIN {X 7.789, Y -16.360, Z 51.000}
   LaserStart_Ext()
   LIN {X 2.424, Y -16.360, Z 51.000}
   LaserEnd_Ext()
   LIN {X -4.674, Y -16.360, Z 51.000}
   LaserStart_Ext()
   LIN {X -7.749, Y -16.360, Z 51.000}
   LaserEnd_Ext()
   LIN {X -7.294, Y -15.360, Z 51.000}
   LaserStart_Ext()
   LIN {X -2.463, Y -15.360, Z 51.000}
   LaserEnd_Ext()
   LIN {X 0.443, Y -15.360, Z 51.000}
   LaserStart_Ext()
   LIN {X 7.917, Y -15.360, Z 51.000}
   LaserEnd_Ext()
   LIN {X 8.044, Y -14.360, Z 51.000}
   LaserStart_Ext()
   LIN {X -6.872, Y -14.360, Z 51.000}
   LaserEnd_Ext()
   LIN {X -6.473, Y -13.360, Z 51.000}
   LaserStart_Ext()
   LIN {X 8.167, Y -13.360, Z 51.000}
   LaserEnd_Ext()
   LIN {X 8.271, Y -12.360, Z 51.000}
   LaserStart_Ext()
   LIN {X -6.072, Y -12.360, Z 51.000}
   LaserEnd_Ext()
   LIN {X -5.669, Y -11.360, Z 51.000}
   LaserStart_Ext()
   LIN {X 8.355, Y -11.360, Z 51.000}
   LaserEnd_Ext()
   LIN {X 8.439, Y -10.360, Z 51.000}
   LaserStart_Ext()
   LIN {X -5.315, Y -10.360, Z 51.000}
   LaserEnd_Ext()
   LIN {X -4.981, Y -9.360, Z 51.000}
   LaserStart_Ext()
   LIN {X 8.526, Y -9.360, Z 51.000}
   LaserEnd_Ext()
   LIN {X 8.614, Y -8.360, Z 51.000}
   LaserStart_Ext()
   LIN {X -4.647, Y -8.360, Z 51.000}
   LaserEnd_Ext()
   LIN {X -4.313, Y -7.360, Z 51.000}
   LaserStart_Ext()
   LIN {X 8.669, Y -7.360, Z 51.000}
   LaserEnd_Ext()
   LIN {X 8.708, Y -6.360, Z 51.000}
   LaserStart_Ext()
   LIN {X -4.009, Y -6.360, Z 51.000}
   LaserEnd_Ext()
   LIN {X -3.743, Y -5.360, Z 51.000}
   LaserStart_Ext()
   LIN {X 8.742, Y -5.360, Z 51.000}
   LaserEnd_Ext()
   LIN {X 8.775, Y -4.360, Z 51.000}
   LaserStart_Ext()
   LIN {X -3.477, Y -4.360, Z 51.000}
   LaserEnd_Ext()
   LIN {X -3.211, Y -3.360, Z 51.000}
   LaserStart_Ext()
   LIN {X 8.808, Y -3.360, Z 51.000}
   LaserEnd_Ext()
   LIN {X 8.841, Y -2.360, Z 51.000}
   LaserStart_Ext()
   LIN {X -2.945, Y -2.360, Z 51.000}
   LaserEnd_Ext()
   LIN {X -2.751, Y -1.360, Z 51.000}
   LaserStart_Ext()
   LIN {X 8.840, Y -1.360, Z 51.000}
   LaserEnd_Ext()
   LIN {X 8.804, Y -0.360, Z 51.000}
   LaserStart_Ext()
   LIN {X -2.565, Y -0.360, Z 51.000}
   LaserEnd_Ext()
   LIN {X -2.380, Y 0.640, Z 51.000}
   LaserStart_Ext()
   LIN {X 8.764, Y 0.640, Z 51.000}
   LaserEnd_Ext()
   LIN {X 8.752, Y 1.640, Z 51.000}
   LaserStart_Ext()
   LIN {X -2.195, Y 1.640, Z 51.000}
   LaserEnd_Ext()
   LIN {X -2.008, Y 2.640, Z 51.000}
   LaserStart_Ext()
   LIN {X 8.746, Y 2.640, Z 51.000}
   LaserEnd_Ext()
   LIN {X 8.740, Y 3.640, Z 51.000}
   LaserStart_Ext()
   LIN {X -1.819, Y 3.640, Z 51.000}
   LaserEnd_Ext()
   LIN {X -1.673, Y 4.640, Z 51.000}
   LaserStart_Ext()
   LIN {X 8.709, Y 4.640, Z 51.000}
   LaserEnd_Ext()
   LIN {X 8.601, Y 5.640, Z 51.000}
   LaserStart_Ext()
   LIN {X -1.597, Y 5.640, Z 51.000}
   LaserEnd_Ext()
   LIN {X -1.521, Y 6.640, Z 51.000}
   LaserStart_Ext()
   LIN {X 8.493, Y 6.640, Z 51.000}
   LaserEnd_Ext()
   LIN {X 8.384, Y 7.640, Z 51.000}
   LaserStart_Ext()
   LIN {X -1.444, Y 7.640, Z 51.000}
   LaserEnd_Ext()
   LIN {X -1.366, Y 8.640, Z 51.000}
   LaserStart_Ext()
   LIN {X 8.276, Y 8.640, Z 51.000}
   LaserEnd_Ext()
   LIN {X 8.168, Y 9.640, Z 51.000}
   LaserStart_Ext()
   LIN {X -1.288, Y 9.640, Z 51.000}
   LaserEnd_Ext()
   LIN {X -1.211, Y 10.640, Z 51.000}
   LaserStart_Ext()
   LIN {X 8.060, Y 10.640, Z 51.000}
   LaserEnd_Ext()
   LIN {X 7.952, Y 11.640, Z 51.000}
   LaserStart_Ext()
   LIN {X -1.128, Y 11.640, Z 51.000}
   LaserEnd_Ext()
   LIN {X -1.028, Y 12.640, Z 51.000}
   LaserStart_Ext()
   LIN {X 7.844, Y 12.640, Z 51.000}
   LaserEnd_Ext()
   LIN {X 7.736, Y 13.640, Z 51.000}
   LaserStart_Ext()
   LIN {X -1.065, Y 13.640, Z 51.000}
   LaserEnd_Ext()
   LIN {X -1.106, Y 14.640, Z 51.000}
   LaserStart_Ext()
   LIN {X 7.638, Y 14.640, Z 51.000}
   LaserEnd_Ext()
   LIN {X 7.541, Y 15.640, Z 51.000}
   LaserStart_Ext()
   LIN {X -1.153, Y 15.640, Z 51.000}
   LaserEnd_Ext()
   LIN {X -1.211, Y 16.640, Z 51.000}
   LaserStart_Ext()
   LIN {X 7.382, Y 16.640, Z 51.000}
   LaserEnd_Ext()
   LIN {X 7.191, Y 17.640, Z 51.000}
   LaserStart_Ext()
   LIN {X -1.269, Y 17.640, Z 51.000}
   LaserEnd_Ext()
   LIN {X -1.327, Y 18.640, Z 51.000}
   LaserStart_Ext()
   LIN {X 7.001, Y 18.640, Z 51.000}
   LaserEnd_Ext()
   LIN {X 6.795, Y 19.640, Z 51.000}
   LaserStart_Ext()
   LIN {X -1.385, Y 19.640, Z 51.000}
   LaserEnd_Ext()
   LIN {X -1.443, Y 20.640, Z 51.000}
   LaserStart_Ext()
   LIN {X 6.585, Y 20.640, Z 51.000}
   LaserEnd_Ext()
   LIN {X 6.376, Y 21.640, Z 51.000}
   LaserStart_Ext()
   LIN {X -1.501, Y 21.640, Z 51.000}
   LaserEnd_Ext()
   LIN {X -1.559, Y 22.640, Z 51.000}
   LaserStart_Ext()
   LIN {X 6.166, Y 22.640, Z 51.000}
   LaserEnd_Ext()
   LIN {X 5.957, Y 23.640, Z 51.000}
   LaserStart_Ext()
   LIN {X -1.617, Y 23.640, Z 51.000}
   LaserEnd_Ext()
   LIN {X -1.733, Y 24.640, Z 51.000}
   LaserStart_Ext()
   LIN {X 5.748, Y 24.640, Z 51.000}
   LaserEnd_Ext()
   LIN {X 5.538, Y 25.640, Z 51.000}
   LaserStart_Ext()
   LIN {X -1.883, Y 25.640, Z 51.000}
   LaserEnd_Ext()
   LIN {X -2.036, Y 26.640, Z 51.000}
   LaserStart_Ext()
   LIN {X 5.257, Y 26.640, Z 51.000}
   LaserEnd_Ext()
   LIN {X 4.972, Y 27.640, Z 51.000}
   LaserStart_Ext()
   LIN {X -2.216, Y 27.640, Z 51.000}
   LaserEnd_Ext()
   LIN {X -2.401, Y 28.640, Z 51.000}
   LaserStart_Ext()
   LIN {X 4.677, Y 28.640, Z 51.000}
   LaserEnd_Ext()
   LIN {X 4.383, Y 29.640, Z 51.000}
   LaserStart_Ext()
   LIN {X -2.606, Y 29.640, Z 51.000}
   LaserEnd_Ext()
   LIN {X -2.831, Y 30.640, Z 51.000}
   LaserStart_Ext()
   LIN {X 4.088, Y 30.640, Z 51.000}
   LaserEnd_Ext()
   LIN {X 3.794, Y 31.640, Z 51.000}
   LaserStart_Ext()
   LIN {X -3.055, Y 31.640, Z 51.000}
   LaserEnd_Ext()
   LIN {X -3.301, Y 32.640, Z 51.000}
   LaserStart_Ext()
   LIN {X 3.505, Y 32.640, Z 51.000}
   LaserEnd_Ext()
   LIN {X 3.192, Y 33.640, Z 51.000}
   LaserStart_Ext()
   LIN {X -3.565, Y 33.640, Z 51.000}
   LaserEnd_Ext()
   LIN {X -3.834, Y 34.640, Z 51.000}
   LaserStart_Ext()
   LIN {X 2.844, Y 34.640, Z 51.000}
   LaserEnd_Ext()
   LIN {X 2.500, Y 35.640, Z 51.000}
   LaserStart_Ext()
   LIN {X -4.132, Y 35.640, Z 51.000}
   LaserEnd_Ext()
   LIN {X -4.431, Y 36.640, Z 51.000}
   LaserStart_Ext()
   LIN {X 2.140, Y 36.640, Z 51.000}
   LaserEnd_Ext()
   LIN {X 1.763, Y 37.640, Z 51.000}
   LaserStart_Ext()
   LIN {X -4.757, Y 37.640, Z 51.000}
   LaserEnd_Ext()
   LIN {X -5.091, Y 38.640, Z 51.000}
   LaserStart_Ext()
   LIN {X 1.389, Y 38.640, Z 51.000}
   LaserEnd_Ext()
   LIN {X 0.992, Y 39.640, Z 51.000}
   LaserStart_Ext()
   LIN {X -5.395, Y 39.640, Z 51.000}
   LaserEnd_Ext()
   LIN {X -5.502, Y 40.640, Z 51.000}
   LaserStart_Ext()
   LIN {X 0.587, Y 40.640, Z 51.000}
   LaserEnd_Ext()
   LIN {X 0.143, Y 41.640, Z 51.000}
   LaserStart_Ext()
   LIN {X -5.247, Y 41.640, Z 51.000}
   LaserEnd_Ext()
   LIN {X -4.453, Y 42.640, Z 51.000}
   LaserStart_Ext()
   LIN {X -0.636, Y 42.640, Z 51.000}
   LaserEnd_Ext()
   LIN {X -5.124, Y -18.157, Z 51.850}
   LaserStart_Ext()
   LIN {X -5.008, Y -18.051, Z 51.850} C_DIS
   LIN {X -3.581, Y -16.739, Z 51.850} C_DIS
   LIN {X -2.295, Y -16.326, Z 51.850} C_DIS
   LIN {X -1.469, Y -16.063, Z 51.850} C_DIS
   LIN {X -0.342, Y -16.204, Z 51.850} C_DIS
   LIN {X 0.675, Y -16.335, Z 51.850} C_DIS
   LIN {X 1.385, Y -16.787, Z 51.850} C_DIS
   LIN {X 2.470, Y -17.472, Z 51.850} C_DIS
   LIN {X 3.255, Y -18.797, Z 51.850} C_DIS
   LIN {X 3.764, Y -19.661, Z 51.850} C_DIS
   LIN {X 3.747, Y -20.772, Z 51.850} C_DIS
   LIN {X 3.771, Y -22.307, Z 51.850} C_DIS
   LIN {X 3.252, Y -23.490, Z 51.850} C_DIS
   LIN {X 3.112, Y -23.786, Z 51.850} C_DIS
   LIN {X 2.951, Y -23.967, Z 51.850} C_DIS
   LIN {X 1.664, Y -25.208, Z 51.850} C_DIS
   LIN {X -0.467, Y -25.930, Z 51.850} C_DIS
   LIN {X -0.685, Y -26.029, Z 51.850} C_DIS
   LIN {X -1.063, Y -25.992, Z 51.850} C_DIS
   LIN {X -2.798, Y -25.754, Z 51.850} C_DIS
   LIN {X -3.873, Y -25.082, Z 51.850} C_DIS
   LIN {X -4.548, Y -24.655, Z 51.850} C_DIS
   LIN {X -5.116, Y -23.810, Z 51.850} C_DIS
   LIN {X -5.712, Y -22.928, Z 51.850} C_DIS
   LIN {X -5.896, Y -21.841, Z 51.850} C_DIS
   LIN {X -6.057, Y -20.870, Z 51.850} C_DIS
   LIN {X -5.243, Y -18.503, Z 51.850} C_DIS
   LIN {X -5.124, Y -18.157, Z 51.850}
   LaserEnd_Ext()
   LIN {X -1.227, Y 44.232, Z 51.850}
   LaserStart_Ext()
   LIN {X 0.150, Y 43.324, Z 51.850} C_DIS
   LIN {X 0.277, Y 43.195, Z 51.850} C_DIS
   LIN {X 1.039, Y 42.047, Z 51.850} C_DIS
   LIN {X 1.479, Y 40.993, Z 51.850} C_DIS
   LIN {X 1.610, Y 40.677, Z 51.850} C_DIS
   LIN {X 1.830, Y 40.127, Z 51.850} C_DIS
   LIN {X 2.222, Y 39.151, Z 51.850} C_DIS
   LIN {X 2.646, Y 38.046, Z 51.850} C_DIS
   LIN {X 3.007, Y 37.088, Z 51.850} C_DIS
   LIN {X 3.431, Y 35.924, Z 51.850} C_DIS
   LIN {X 4.199, Y 33.696, Z 51.850} C_DIS
   LIN {X 4.376, Y 33.163, Z 51.850} C_DIS
   LIN {X 5.668, Y 28.777, Z 51.850} C_DIS
   LIN {X 6.531, Y 25.750, Z 51.850} C_DIS
   LIN {X 7.763, Y 19.865, Z 51.850} C_DIS
   LIN {X 8.600, Y 15.474, Z 51.850} C_DIS
   LIN {X 8.926, Y 12.100, Z 51.850} C_DIS
   LIN {X 9.758, Y 4.399, Z 51.850} C_DIS
   LIN {X 9.775, Y 1.487, Z 51.850} C_DIS
   LIN {X 9.818, Y 0.401, Z 51.850} C_DIS
   LIN {X 9.891, Y -1.680, Z 51.850} C_DIS
   LIN {X 9.722, Y -6.787, Z 51.850} C_DIS
   LIN {X 9.685, Y -8.058, Z 51.850} C_DIS
   LIN {X 9.647, Y -8.546, Z 51.850} C_DIS
   LIN {X 9.287, Y -12.830, Z 51.850} C_DIS
   LIN {X 9.001, Y -15.214, Z 51.850} C_DIS
   LIN {X 8.824, Y -16.608, Z 51.850} C_DIS
   LIN {X 8.615, Y -17.935, Z 51.850} C_DIS
   LIN {X 8.373, Y -19.534, Z 51.850} C_DIS
   LIN {X 8.092, Y -21.106, Z 51.850} C_DIS
   LIN {X 7.788, Y -22.745, Z 51.850} C_DIS
   LIN {X 6.828, Y -24.959, Z 51.850} C_DIS
   LIN {X 6.287, Y -26.223, Z 51.850} C_DIS
   LIN {X 5.563, Y -26.895, Z 51.850} C_DIS
   LIN {X 3.835, Y -28.572, Z 51.850} C_DIS
   LIN {X 1.153, Y -29.639, Z 51.850} C_DIS
   LIN {X 0.299, Y -29.948, Z 51.850} C_DIS
   LIN {X -0.872, Y -29.748, Z 51.850} C_DIS
   LIN {X -5.431, Y -28.958, Z 51.850} C_DIS
   LIN {X -6.255, Y -28.319, Z 51.850} C_DIS
   LIN {X -7.720, Y -27.166, Z 51.850} C_DIS
   LIN {X -9.353, Y -24.391, Z 51.850} C_DIS
   LIN {X -9.619, Y -23.933, Z 51.850} C_DIS
   LIN {X -9.686, Y -23.308, Z 51.850} C_DIS
   LIN {X -10.032, Y -20.245, Z 51.850} C_DIS
   LIN {X -9.251, Y -17.443, Z 51.850} C_DIS
   LIN {X -9.180, Y -17.192, Z 51.850} C_DIS
